# B&R Automation Studio project brdkViLibs
Automation Studio 4.9.4.92 SP; technology packages: mapp 5.20.0, mappView 5.20.0, mappVision 5.20.0

## Configuration ARM

CPU X90CP174.24-00, AutomationRuntime C4.90, Build 6.3.0, Safety 0.0, Vc V4.72.2

CPU X20CP0483, AutomationRuntime C4.90, Build 6.3.0, Safety 0.0, Vc V4.72.2

CPU X20CP0484-1, AutomationRuntime C4.90, Build 6.3.0, Safety 0.0, Vc V4.72.2

### Task classes (Cpu.sw)
```
Cyclic#2 (cycle 20000 us, tolerance 20000 us):
  Demo <- Demo.prg
  Recipe <- Recipe.prg
Binaries: udbdef, mvLoader, TCData, FWRules, TCLang, visionUnit, ashwac, Settings, User, sysconf, viComp, asfw, arconfig, ashwd, iomap, Role, viApp, Config, px, TC, arflatprv, arcoal, arsvcreg, mCoWebSc, Settings_1
Libraries: ViBase, MpRecipe, MpBase, runtime, astime, AsZip, FileIO, AsARCfg, powerlnk, AsEPL, AsIO, sys_lib, standard, MTLinAlg, brdkViMapp, brdkViImg, brdkViGeom, brdkViBase, brdkViVF, brdkViCal, AsTCP, brsystem, AsHttp, AsIecCon, asbrstr, asiodiag, arssl
```

### Task classes (Cpu.sw)
```
Cyclic#1 (cycle 1000 us, tolerance 10000 us):
  Recipe <- Recipe.prg
  Calibratio <- Calibration.prg
Binaries: udbdef, mvLoader, TCData, FWRules, TCLang, ashwac, Settings, User, sysconf, viComp, asfw, arconfig, ashwd, iomap, Role, viApp, Config, px, TC, arflatprv, arcoal, arsvcreg
Libraries: ViBase, MpRecipe, MpBase, runtime, astime, AsZip, FileIO, AsARCfg, powerlnk, AsEPL, AsIO, sys_lib, AsHttp, standard, MTLinAlg, brdkViMapp, brdkViBase, brdkViVF, BRSE_RTK, brdkViCal, brdkViImg, asieccon, brdkViGeom
```

### Task classes (Cpu.sw)
```
Cyclic#1 (cycle 1000 us, tolerance 10000 us):
  Recipe <- Recipe.prg
  Calibratio <- Calibration.prg
Binaries: udbdef, mvLoader, TCData, FWRules, TCLang, ashwac, Settings, User, sysconf, viComp, asfw, arconfig, ashwd, iomap, Role, viApp, Config, px, TC, arflatprv, arcoal, arsvcreg
Libraries: ViBase, MpRecipe, MpBase, brdkViGeom, runtime, astime, AsZip, FileIO, AsARCfg, powerlnk, AsEPL, AsIO, sys_lib, AsHttp, standard, brdkViImg, MTLinAlg, brdkViMapp, AsIODiag, brdkViBase, brdkViVF, BRSE_RTK, brdkViCal, asieccon
```

### Hardware
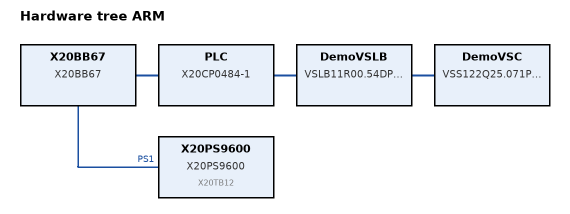
```
DemoVSC : VSS122Q25.071P-000 v1.7.0.606  [PLK1 -> DemoVSLB.PLK2 (NodeNumber=6) [Cable Type=PowerlinkCable, Length=10, Version=1.0.0.3]]
  Supervision = off
  VisionConfig = gBlobCamera
DemoVSLB : VSLB11R00.54DP-000 v1.1.0.323  [PLK1 -> PLC.IF3 (NodeNumber=2) [Cable Type=PowerlinkCable, Length=10, Version=1.0.0.3]; PLK2 -> DemoVSC.PLK1 (NodeNumber=2) [Cable Type=PowerlinkCable, Length=10, Version=1.0.0.3]]
  Supervision = off
  VisionConfig = gBlobCamera
PLC : X20CP0484-1 v1.7.0.0  [SL -> X20BB67.SL1]
  Connector IF2:
    ActivateDevice = 1
    Mode = Manual
    InternetAddress = 192.168.87.210
    SubnetMask = 255.255.255.0
  Connector IF3:
    MtuSize = 1500
    DNAConfiguration = manual
    CycleTime = 1000
    AsyncTimeout = 20
    AsyncSlotsPerCycle = 7
    InternetAddress = 192.168.200.240
    SubnetMask = 255.255.255.0
  ConfigurationID = brdkVision
  UserPartitionSize = 100
  TimerDeviceType = EPLX2X
  TimerDevice = PLC.IF3
  IdleTaskClass = 4
  TaskClassIdleTime = 2000
  Cyclic1Duration = 1000
  Cyclic1Tolerance = 10000
  Cyclic1Stack = 1000000
  Cyclic2Duration = 20000
  Cyclic2Tolerance = 20000
  Cyclic3Duration = 50000
  Cyclic3Tolerance = 50000
  Cyclic4Duration = 100000
  Cyclic4Tolerance = 100000
  Cyclic5Duration = 200000
  Cyclic5Tolerance = 200000
  Cyclic6Duration = 500000
  Cyclic6Tolerance = 500000
  Cyclic7Duration = 1000000
  Cyclic7Tolerance = 1000000
  Cyclic8Duration = 10000
  Cyclic8Tolerance = 30000000
  FileDevice1
  FileDeviceName1 = RECIPE
  FileDevicePath1 = F:\
  FileDevice2
  FileDeviceName2 = SIM
  FileDevicePath2 = C:\simPlc\brdkVision
  FtpUser1
  FtpUsername1 = admin
  FtpUserPassword1 = 4WFXWDK5TMVpfeai37B+7WhwHoefN0SDX+8eS6SXEy0=
  FtpUserSalt1 = PfytuFsU
  FTPAccessRight1 = 0
  FTPdevice1 = ALL
  ActivateOpcUa = 1
  OpcUaInformationModels_PV_Version = 1
X20BB67 : X20BB67 v1.2.0.0
X20PS9600 : X20PS9600 v1.6.0.0  [PS -> X20BB67.PS1; SS1 -> X20TB12.SS]
X20TB12 : X20TB12 v1.0.0.0
```

### Cpu.sw.bak1 - PLC/Cpu.sw.bak1
```
SwConfiguration (CpuAddress=SL1)
  TaskClass Cyclic#1
  TaskClass Cyclic#2:
    Task Demo (Source=Demo.prg, Memory=UserROM, Language=IEC, Debugging=true)
    Task Recipe (Source=Recipe.prg, Memory=UserROM, Language=IEC, Debugging=true)
  TaskClass Cyclic#3
  TaskClass Cyclic#4
  TaskClass Cyclic#5
  TaskClass Cyclic#6
  TaskClass Cyclic#7
  TaskClass Cyclic#8
  Binaries:
    BinaryObject udbdef (Source=, Memory=UserROM, Language=Binary)
    BinaryObject mvLoader (Source=, Memory=UserROM, Language=Binary)
    BinaryObject TCData (Source=, Memory=SystemROM, Language=Binary)
    BinaryObject FWRules (Source=, Memory=UserROM, Language=Binary)
    BinaryObject TCLang (Source=, Memory=UserROM, Language=Binary)
    BinaryObject visionUnit (Source=, Memory=UserROM, Language=Binary)
    BinaryObject arflatprv (Source=, Memory=UserROM, Language=Binary)
    BinaryObject arcoal (Source=, Memory=UserROM, Language=Binary)
    BinaryObject arsvcreg (Source=, Memory=UserROM, Language=Binary)
    BinaryObject mCoWebSc (Source=, Memory=UserROM, Language=Binary)
    BinaryObject ashwac (Source=, Memory=UserROM, Language=Binary)
    BinaryObject Settings (Source=, Memory=UserROM, Language=Binary)
    BinaryObject User (Source=, Memory=UserROM, Language=Binary)
    BinaryObject sysconf (Source=, Memory=SystemROM, Language=Binary)
    BinaryObject viComp (Source=, Memory=UserROM, Language=Binary)
    BinaryObject asfw (Source=, Memory=SystemROM, Language=Binary)
    BinaryObject arconfig (Source=, Memory=SystemROM, Language=Binary)
    BinaryObject ashwd (Source=, Memory=SystemROM, Language=Binary)
    BinaryObject iomap (Source=, Memory=UserROM, Language=Binary)
    BinaryObject Role (Source=, Memory=UserROM, Language=Binary)
    BinaryObject viApp (Source=, Memory=UserROM, Language=Binary)
    BinaryObject Config (Source=, Memory=UserROM, Language=Binary)
    BinaryObject px (Source=, Memory=UserROM, Language=Binary)
    BinaryObject TC (Source=, Memory=UserROM, Language=Binary)
    BinaryObject Settings_1 (Source=, Memory=UserROM, Language=Binary)
  Libraries:
    LibraryObject ViBase (Source=Libraries.ViBase.lby, Memory=UserROM, Language=binary, Debugging=true)
    LibraryObject MpRecipe (Source=Libraries.MpRecipe.lby, Memory=UserROM, Language=Binary, Debugging=true)
    LibraryObject MpBase (Source=Libraries.MpBase.lby, Memory=UserROM, Language=Binary, Debugging=true)
    LibraryObject runtime (Source=Libraries.runtime.lby, Memory=UserROM, Language=binary, Debugging=true)
    LibraryObject astime (Source=Libraries.astime.lby, Memory=UserROM, Language=binary, Debugging=true)
    LibraryObject AsZip (Source=Libraries.AsZip.lby, Memory=UserROM, Language=binary, Debugging=true)
    LibraryObject FileIO (Source=Libraries.FileIO.lby, Memory=UserROM, Language=binary, Debugging=true)
    LibraryObject AsARCfg (Source=Libraries.AsARCfg.lby, Memory=UserROM, Language=binary, Debugging=true)
    LibraryObject powerlnk (Source=Libraries.powerlnk.lby, Memory=UserROM, Language=binary, Debugging=true)
    LibraryObject AsEPL (Source=Libraries.AsEPL.lby, Memory=UserROM, Language=binary, Debugging=true)
    LibraryObject AsIO (Source=Libraries.AsIO.lby, Memory=UserROM, Language=binary, Debugging=true)
    LibraryObject sys_lib (Source=Libraries.sys_lib.lby, Memory=UserROM, Language=binary, Debugging=true)
    LibraryObject standard (Source=Libraries.standard.lby, Memory=UserROM, Language=binary, Debugging=true)
    LibraryObject MTLinAlg (Source=Libraries.MTLinAlg.lby, Memory=UserROM, Language=Binary, Debugging=true)
    LibraryObject brdkViMapp (Source=Libraries.brdkViLibs.brdkViMapp.lby, Memory=UserROM, Language=Binary, Debugging=true)
    LibraryObject brdkViImg (Source=Libraries.brdkViLibs.brdkViImg.lby, Memory=UserROM, Language=Binary, Debugging=true)
    LibraryObject brdkViGeom (Source=Libraries.brdkViLibs.brdkViGeom.lby, Memory=UserROM, Language=Binary, Debugging=true)
    LibraryObject brdkViBase (Source=Libraries.brdkViLibs.brdkViBase.lby, Memory=UserROM, Language=Binary, Debugging=true)
    LibraryObject brdkViVF (Source=Libraries.brdkViLibs.brdkViVF.lby, Memory=UserROM, Language=Binary, Debugging=true)
    LibraryObject brdkViCal (Source=Libraries.brdkViLibs.brdkViCal.lby, Memory=UserROM, Language=Binary, Debugging=true)
    LibraryObject AsTCP (Source=Libraries.AsTCP.lby, Memory=UserROM, Language=binary, Debugging=true)
    LibraryObject brsystem (Source=Libraries.brsystem.lby, Memory=UserROM, Language=binary, Debugging=true)
    LibraryObject AsHttp (Source=Libraries.AsHttp.lby, Memory=UserROM, Language=binary, Debugging=true)
    LibraryObject JSON_WS (Source=Libraries.brdkViLibs.JSON_WS.lby, Memory=UserROM, Language=ANSIC, Debugging=true)
    LibraryObject AsIecCon (Source=Libraries.AsIecCon.lby, Memory=UserROM, Language=binary, Debugging=true)
    LibraryObject arssl (Source=, Memory=UserROM, Language=Binary, Debugging=true)
    LibraryObject asbrstr (Source=, Memory=UserROM, Language=Binary, Debugging=true)
    LibraryObject asiodiag (Source=, Memory=UserROM, Language=Binary, Debugging=true)
```

### IoMap.iom - PLC/IoMap.iom
```iecst
VAR_CONFIG
	::Demo:hw.cam.in.common.moduleOk AT %IX."DemoVSC".ModuleOk;
	::Demo:hw.cam.in.common.serialNumber AT %ID."DemoVSC".SerialNumber;
	::Demo:hw.cam.in.common.moduleId AT %ID."DemoVSC".ModuleID;
	::Demo:hw.cam.in.common.hardwareVariant AT %ID."DemoVSC".HardwareVariant;
	::Demo:hw.cam.in.common.firmwareVersion AT %ID."DemoVSC".FirmwareVersion;
	::Demo:hw.cam.in.status.sensorTemperature AT %IB."DemoVSC".SensorTemperature;
	::Demo:hw.cam.in.status.lightWarningCnt AT %IB."DemoVSC".LightWarningCnt;
	::Demo:hw.cam.in.status.cameraStatus AT %ID."DemoVSC".CameraStatus;
	::Demo:hw.cam.in.status.acceptedAcquisitionCnt AT %IB."DemoVSC".AcceptedAcquisitionCnt;
	::Demo:hw.cam.in.status.completedAcquisitionCnt AT %IB."DemoVSC".CompletedAcquisitionCnt;
	::Demo:hw.cam.in.status.failedAcquisitionCnt AT %IB."DemoVSC".FailedAcquisitionCnt;
	::Demo:hw.cam.in.status.gainLevel AT %IB."DemoVSC".ReadGainLevel;
	::Demo:hw.cam.in.status.focus AT %IW."DemoVSC".ReadFocus;
	::Demo:hw.cam.in.status.exposureTime AT %ID."DemoVSC".ReadExposureTime;
	::Demo:hw.cam.in.status.undervoltageError AT %IX."DemoVSC".UndervoltageError;
	::Demo:hw.cam.in.status.digitalInput AT %IX."DemoVSC".DigitalInput01;
	::Demo:hw.cam.in.status.digitalOutputStatus AT %IX."DemoVSC".DigitalOutputStatus01;
	::Demo:hw.cam.in.status.imageAcquisitionReady AT %IX."DemoVSC".ImageAcquisitionReady;
	::Demo:hw.cam.in.status.imageProcessingActive AT %IX."DemoVSC".ImageProcessingActive;
	::Demo:hw.cam.in.status.cameraProcessingTime AT %IW."DemoVSC".CameraProcessingTime;
	::Demo:hw.cam.in.status.imageProcessingError AT %IW."DemoVSC".ImageProcessingError;
	::Demo:hw.cam.in.status.imageNettime AT %ID."DemoVSC".ImageNettime;
	::Demo:hw.cam.out.par.statusLED AT %QB."DemoVSC".StatusLED;
	::Demo:hw.cam.out.par.gainLevel AT %QB."DemoVSC".GainLevel;
	::Demo:hw.cam.out.par.focus AT %QW."DemoVSC".SetFocus;
	::Demo:hw.cam.out.par.exposureTime AT %QD."DemoVSC".ExposureTime01;
	::Demo:hw.cam.out.par.delayNetTime AT %QD."DemoVSC".DelayNettime01;
	::Demo:hw.cam.out.par.flashColor AT %QB."DemoVSC".FlashColor01;
	::Demo:hw.cam.out.par.flashSegment AT %QB."DemoVSC".FlashSegment01;
	::Demo:hw.cam.out.cmd.digitalOutput AT %QX."DemoVSC".DigitalOutput01;
	::Demo:hw.cam.out.par.IRFilter AT %QX."DemoVSC".IRFilter;
	::Demo:hw.cam.out.par.chromaticLock AT %QX."DemoVSC".ChromaticLock;
	::Demo:hw.cam.out.cmd.searchAcquisitonSettings AT %QX."DemoVSC".SearchAcquisitionSettings;
	::Demo:hw.cam.out.cmd.resetAcquisiton AT %QX."DemoVSC".ResetAcquisition;
	::Demo:hw.cam.out.cmd.imageAcquisition AT %QX."DemoVSC".ImageAcquisition;
	::Demo:hw.blob.out.common.enable AT %QX."DemoVSC".Enable_1;
	::Demo:hw.blob.out.common.numSearchMax AT %QB."DemoVSC".NumSearchMax_1;
	::Demo:hw.blob.out.regionFeatures AT %QX."DemoVSC".RegionFeatures_1;
	::Demo:hw.blob.out.enhancedBlobInformation AT %QX."DemoVSC".EnhancedBlobInformation_1;
	::Demo:hw.blob.out.common.alignment AT %QB."DemoVSC".Alignment_1;
	::Demo:hw.blob.out.common.offsetROI.x AT %QD."DemoVSC".OffsetROIX_1;
	::Demo:hw.blob.out.common.offsetROI.y AT %QD."DemoVSC".OffsetROIY_1;
	::Demo:hw.blob.out.common.offsetROI.orientation AT %QW."DemoVSC".OffsetROIOrientation_1;
	::Demo:hw.blob.out.common.offsetROI.x AT %QD."DemoVSC".OffsetROIRotCenterX_1;
	::Demo:hw.blob.out.common.offsetROI.y AT %QD."DemoVSC".OffsetROIRotCenterY_1;
	::Demo:hw.blob.in.common.numResults AT %IB."DemoVSC".NumResults_1;
	::Demo:hw.blob.in.common.functionProcessingTime AT %IW."DemoVSC".FunctionProcessingTime_1;
	::Demo:hw.blob.in.results[0].modelNumber AT %IB."DemoVSC".ModelNumber_101;
	::Demo:hw.blob.in.results[0].meanGreyValue AT %IB."DemoVSC".MeanGrayValue_101;
	::Demo:hw.blob.in.results[0].clipped AT %IX."DemoVSC".Clipped_101;
	::Demo:hw.blob.in.results[0].area AT %ID."DemoVSC".Area_101;
	::Demo:hw.blob.in.results[0].length AT %ID."DemoVSC".Length_101;
	::Demo:hw.blob.in.results[0].width AT %ID."DemoVSC".Width_101;
	::Demo:hw.blob.in.results[0].xMin AT %ID."DemoVSC".Xmin_101;
	::Demo:hw.blob.in.results[0].xMax AT %ID."DemoVSC".Xmax_101;
	::Demo:hw.blob.in.results[0].yMin AT %ID."DemoVSC".Ymin_101;
	::Demo:hw.blob.in.results[0].yMax AT %ID."DemoVSC".Ymax_101;
	::Demo:hw.blob.in.results[0].circularity AT %IB."DemoVSC".Circularity_101;
	::Demo:hw.blob.in.results[0].rectangularity AT %IB."DemoVSC".Rectangularity_101;
	::Demo:hw.blob.in.results[0].anisometry AT %IW."DemoVSC".Anisometry_101;
	::Demo:hw.blob.in.results[0].innterCirclePositionX AT %ID."DemoVSC".InnerCirclePositionX_101;
	::Demo:hw.blob.in.results[0].innterCirclePositionY AT %ID."DemoVSC".InnerCirclePositionY_101;
	::Demo:hw.blob.in.results[0].innterCircleRadius AT %ID."DemoVSC".InnerCircleRadius_101;
	::Demo:hw.blob.in.results[0].positionX AT %ID."DemoVSC".PositionX_101;
	::Demo:hw.blob.in.results[0].positionY AT %ID."DemoVSC".PositionY_101;
	::Demo:hw.blob.in.results[0].orientation AT %IW."DemoVSC".Orientation_101;
	::Demo:hw.blob.in.results[0].rotCenterX AT %ID."DemoVSC".RotCenterX_101;
	::Demo:hw.blob.in.results[0].rotCenterY AT %ID."DemoVSC".RotCenterY_101;
	::Demo:hw.blob.in.results[1].modelNumber AT %IB."DemoVSC".ModelNumber_102;
	::Demo:hw.blob.in.results[1].meanGreyValue AT %IB."DemoVSC".MeanGrayValue_102;
	::Demo:hw.blob.in.results[1].clipped AT %IX."DemoVSC".Clipped_102;
	::Demo:hw.blob.in.results[1].area AT %ID."DemoVSC".Area_102;
	::Demo:hw.blob.in.results[1].length AT %ID."DemoVSC".Length_102;
	::Demo:hw.blob.in.results[1].width AT %ID."DemoVSC".Width_102;
	::Demo:hw.blob.in.results[1].xMin AT %ID."DemoVSC".Xmin_102;
	::Demo:hw.blob.in.results[1].xMax AT %ID."DemoVSC".Xmax_102;
	::Demo:hw.blob.in.results[1].yMin AT %ID."DemoVSC".Ymin_102;
	::Demo:hw.blob.in.results[1].yMax AT %ID."DemoVSC".Ymax_102;
	::Demo:hw.blob.in.results[1].circularity AT %IB."DemoVSC".Circularity_102;
	::Demo:hw.blob.in.results[1].rectangularity AT %IB."DemoVSC".Rectangularity_102;
	::Demo:hw.blob.in.results[1].anisometry AT %IW."DemoVSC".Anisometry_102;
	::Demo:hw.blob.in.results[1].innterCirclePositionX AT %ID."DemoVSC".InnerCirclePositionX_102;
	::Demo:hw.blob.in.results[1].innterCirclePositionY AT %ID."DemoVSC".InnerCirclePositionY_102;
	::Demo:hw.blob.in.results[1].innterCircleRadius AT %ID."DemoVSC".InnerCircleRadius_102;
	::Demo:hw.blob.in.results[1].positionX AT %ID."DemoVSC".PositionX_102;
	::Demo:hw.blob.in.results[1].positionY AT %ID."DemoVSC".PositionY_102;
	::Demo:hw.blob.in.results[1].orientation AT %IW."DemoVSC".Orientation_102;
	::Demo:hw.blob.in.results[1].rotCenterX AT %ID."DemoVSC".RotCenterX_102;
	::Demo:hw.blob.in.results[1].rotCenterY AT %ID."DemoVSC".RotCenterY_102;
	::Demo:hw.blob.in.results[2].modelNumber AT %IB."DemoVSC".ModelNumber_103;
	::Demo:hw.blob.in.results[2].meanGreyValue AT %IB."DemoVSC".MeanGrayValue_103;
	::Demo:hw.blob.in.results[2].clipped AT %IX."DemoVSC".Clipped_103;
	::Demo:hw.blob.in.results[2].area AT %ID."DemoVSC".Area_103;
	::Demo:hw.blob.in.results[2].length AT %ID."DemoVSC".Length_103;
	::Demo:hw.blob.in.results[2].width AT %ID."DemoVSC".Width_103;
	::Demo:hw.blob.in.results[2].xMin AT %ID."DemoVSC".Xmin_103;
	::Demo:hw.blob.in.results[2].xMax AT %ID."DemoVSC".Xmax_103;
	::Demo:hw.blob.in.results[2].yMin AT %ID."DemoVSC".Ymin_103;
	::Demo:hw.blob.in.results[2].yMax AT %ID."DemoVSC".Ymax_103;
	::Demo:hw.blob.in.results[2].circularity AT %IB."DemoVSC".Circularity_103;
	::Demo:hw.blob.in.results[2].rectangularity AT %IB."DemoVSC".Rectangularity_103;
	::Demo:hw.blob.in.results[2].anisometry AT %IW."DemoVSC".Anisometry_103;
	::Demo:hw.blob.in.results[2].innterCirclePositionX AT %ID."DemoVSC".InnerCirclePositionX_103;
	::Demo:hw.blob.in.results[2].innterCirclePositionY AT %ID."DemoVSC".InnerCirclePositionY_103;
	::Demo:hw.blob.in.results[2].innterCircleRadius AT %ID."DemoVSC".InnerCircleRadius_103;
	::Demo:hw.blob.in.results[2].positionX AT %ID."DemoVSC".PositionX_103;
	::Demo:hw.blob.in.results[2].positionY AT %ID."DemoVSC".PositionY_103;
	::Demo:hw.blob.in.results[2].orientation AT %IW."DemoVSC".Orientation_103;
	::Demo:hw.blob.in.results[2].rotCenterX AT %ID."DemoVSC".RotCenterX_103;
	::Demo:hw.blob.in.results[2].rotCenterY AT %ID."DemoVSC".RotCenterY_103;
	::Demo:hw.blob.in.results[3].modelNumber AT %IB."DemoVSC".ModelNumber_104;
	::Demo:hw.blob.in.results[3].meanGreyValue AT %IB."DemoVSC".MeanGrayValue_104;
	::Demo:hw.blob.in.results[3].clipped AT %IX."DemoVSC".Clipped_104;
	::Demo:hw.blob.in.results[3].area AT %ID."DemoVSC".Area_104;
	::Demo:hw.blob.in.results[3].length AT %ID."DemoVSC".Length_104;
	::Demo:hw.blob.in.results[3].width AT %ID."DemoVSC".Width_104;
	::Demo:hw.blob.in.results[3].xMin AT %ID."DemoVSC".Xmin_104;
	::Demo:hw.blob.in.results[3].xMax AT %ID."DemoVSC".Xmax_104;
	::Demo:hw.blob.in.results[3].yMin AT %ID."DemoVSC".Ymin_104;
	::Demo:hw.blob.in.results[3].yMax AT %ID."DemoVSC".Ymax_104;
	::Demo:hw.blob.in.results[3].circularity AT %IB."DemoVSC".Circularity_104;
	::Demo:hw.blob.in.results[3].rectangularity AT %IB."DemoVSC".Rectangularity_104;
	::Demo:hw.blob.in.results[3].anisometry AT %IW."DemoVSC".Anisometry_104;
	::Demo:hw.blob.in.results[3].innterCirclePositionX AT %ID."DemoVSC".InnerCirclePositionX_104;
	::Demo:hw.blob.in.results[3].innterCirclePositionY AT %ID."DemoVSC".InnerCirclePositionY_104;
	::Demo:hw.blob.in.results[3].innterCircleRadius AT %ID."DemoVSC".InnerCircleRadius_104;
	::Demo:hw.blob.in.results[3].positionX AT %ID."DemoVSC".PositionX_104;
	::Demo:hw.blob.in.results[3].positionY AT %ID."DemoVSC".PositionY_104;
	::Demo:hw.blob.in.results[3].orientation AT %IW."DemoVSC".Orientation_104;
	::Demo:hw.blob.in.results[3].rotCenterX AT %ID."DemoVSC".RotCenterX_104;
	::Demo:hw.blob.in.results[3].rotCenterY AT %ID."DemoVSC".RotCenterY_104;
	::Demo:hw.io.input.nettime AT %ID."PLC".IF3.NettimeSoC;
	::Demo:hw.backLight[0].in.common.moduleOk AT %IX."DemoVSLB".ModuleOk;
	::Demo:hw.backLight[0].in.common.serialNumber AT %ID."DemoVSLB".SerialNumber;
	::Demo:hw.backLight[0].in.common.moduleId AT %ID."DemoVSLB".ModuleID;
	::Demo:hw.backLight[0].in.common.hardwareVariant AT %ID."DemoVSLB".HardwareVariant;
	::Demo:hw.backLight[0].in.common.firmwareVersion AT %ID."DemoVSLB".FirmwareVersion;
	::Demo:hw.backLight[0].in.status.ready AT %IX."DemoVSLB".Ready;
	::Demo:hw.backLight[0].in.status.status AT %ID."DemoVSLB".Status;
	::Demo:hw.backLight[0].in.status.acceptedFlashCnt AT %IB."DemoVSLB".AcceptedFlashCnt;
	::Demo:hw.backLight[0].in.status.completedFlashCnt AT %IB."DemoVSLB".CompletedFlashCnt;
	::Demo:hw.backLight[0].in.status.failedFlashCnt AT %IB."DemoVSLB".FailedFlashCnt;
	::Demo:hw.backLight[0].in.status.LightWarningCnt AT %IB."DemoVSLB".LightWarningCnt;
	::Demo:hw.backLight[0].in.status.sensorTemperatureControllerBoard AT %IB."DemoVSLB".SensorTemperature;
	::Demo:hw.backLight[0].out.cmd.flashTrigger AT %QX."DemoVSLB".FlashTrigger;
	::Demo:hw.backLight[0].out.cmd.resetFlashTrigger AT %QX."DemoVSLB".ResetFlashTrigger;
	::Demo:hw.backLight[0].out.par.nettime AT %QD."DemoVSLB".Nettime01;
	::Demo:hw.backLight[0].out.par.exposureTime AT %QD."DemoVSLB".ExposureTime01;
	::Demo:hw.backLight[0].out.par.flashColor AT %QB."DemoVSLB".FlashColor01;
END_VAR
```

### Config.mprecipecsv - PLC/mappServices/Config.mprecipecsv
```
Element gRecipeCsv (Type=mprecipecsv)
```

### IoMap.iom - X20CP0483/IoMap.iom
```iecst
VAR_CONFIG
	::Calibratio:hw.out.focus AT %QW."VSC122R14.033P-000".SetFocus;
	::Calibratio:hw.out.expTime AT %QD."VSC122R14.033P-000".ExposureTime01;
	::Calibratio:hw.out.delayNettime AT %QD."VSC122R14.033P-000".DelayNettime01;
	::Calibratio:hw.out.ledColor AT %QB."VSC122R14.033P-000".FlashColor01;
	::Calibratio:hw.out.ledSegment AT %QB."VSC122R14.033P-000".FlashSegment01;
	::Calibratio:hw.in.ready AT %IX."VSC122R14.033P-000".ImageAcquisitionReady;
	::Calibratio:hw.out.trigger AT %QX."VSC122R14.033P-000".ImageAcquisition;
	::Calibratio:hw.out.irFilter AT %QX."VSC122R14.033P-000".IRFilter;
	::Calibratio:hw.out.enable AT %QX."VSC122R14.033P-000".VF1Enable;
	::Calibratio:hw.out.numMax AT %QB."VSC122R14.033P-000".VF1NumSearchMax;
	::Calibratio:hw.in.imgTime AT %ID."VSC122R14.033P-000".ImageNettime;
	::Calibratio:hw.in.va.numRes AT %IB."VSC122R14.033P-000".NumResults;
	::Calibratio:hw.in.va.res[0].posX AT %ID."VSC122R14.033P-000".PositionX01;
	::Calibratio:hw.in.va.res[1].posX AT %ID."VSC122R14.033P-000".PositionX02;
	::Calibratio:hw.in.va.res[2].posX AT %ID."VSC122R14.033P-000".PositionX03;
	::Calibratio:hw.in.va.res[3].posX AT %ID."VSC122R14.033P-000".PositionX04;
	::Calibratio:hw.in.va.res[0].posY AT %ID."VSC122R14.033P-000".PositionY01;
	::Calibratio:hw.in.va.res[1].posY AT %ID."VSC122R14.033P-000".PositionY02;
	::Calibratio:hw.in.va.res[2].posY AT %ID."VSC122R14.033P-000".PositionY03;
	::Calibratio:hw.in.va.res[3].posY AT %ID."VSC122R14.033P-000".PositionY04;
	::Calibratio:hw.out.delayNettime AT %QD."VSLB11Q00.54DP-000".Nettime01;
	::Calibratio:hw.out.expTime AT %QD."VSLB11Q00.54DP-000".ExposureTime01;
	::Calibratio:hw.out.ledColor AT %QB."VSLB11Q00.54DP-000".FlashColor01;
	::Calibratio:hw.out.trigger AT %QX."VSLB11Q00.54DP-000".FlashTrigger;
	::Calibratio:hw.out.useRegionFeat AT %QX."VSC122R14.033P-000".VF1RegionFeatures;
	::Calibratio:hw.in.nettime AT %ID."X20CP0483".IF3.NettimeSoC;
END_VAR
```

### IoMap.iom - X20CP0484_1/IoMap.iom
```iecst
VAR_CONFIG
	::Calibratio:hw.io.input.nettime AT %ID."X20CP0484_1".IF3.NettimeSoC;
END_VAR
```

### Settings.vicfg - X20CP0484_1/mappVision/Settings.vicfg
```
Element VisionSettings (Type=vicfg)
  ActivateVisualization = TRUE
  FileDeviceName
  Permissions:
    WriteAccessRole = Everyone
```

### viComp.visioncomponent - X20CP0484_1/mappVision/viComp.visioncomponent
```
Element gBlobCamera (Type=visioncomponent)
  VisionApplicationReference = BLOBCam
```

## Configuration Intel

CPU X20CP1586, AutomationRuntime C4.90, Build 6.3.0, Safety 0.0, Vc 

CPU X20CP1586, AutomationRuntime C4.90, Build 6.3.0, Safety 0.0, Vc 

### Task classes (Cpu.sw)
```
Cyclic#1 (cycle 2000 us):
  Recipe <- Recipe.prg
  Demo <- Demo.prg
Binaries: udbdef, mvLoader, TCData, FWRules, TCLang, arflatprv, arcoal, arsvcreg, visionUnit, ashwac, Settings, User, sysconf, viComp, asfw, arconfig, ashwd, iomap, Role, viApp, Config
Libraries: ViBase, MpRecipe, MpBase, MTLinAlg, runtime, astime, AsZip, FileIO, AsARCfg, powerlnk, AsEPL, AsIO, sys_lib, standard, brdkViBase, brdkViMapp, brdkViVF, brdkViCal, AsIODiag, arssl, asieccon
```

### Task classes (Cpu.sw)
```
Cyclic#1 (cycle 2000 us):
  Recipe <- Recipe.prg
  Calibratio <- Calibration.prg
Binaries: udbdef, mvLoader, TCData, FWRules, TCLang, ashwac, Settings, User, sysconf, viComp, asfw, arconfig, ashwd, iomap, Role, viApp, Config, arflatprv, arcoal, arsvcreg
Libraries: ViBase, MpRecipe, MpBase, MTLinAlg, runtime, astime, AsZip, FileIO, AsARCfg, powerlnk, AsEPL, AsIO, sys_lib, AsHttp, standard, arssl, brdkViBase, brdkViGeom, brdkViImg, brdkViMapp, brdkViVF, BRSE_RTK, brdkViCal
```

### Hardware
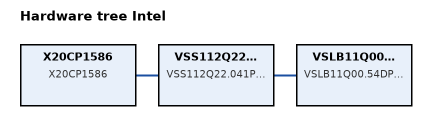
```
VSLB11Q00.54DP-000 : VSLB11Q00.54DP-000 v1.1.0.323  [PLK1 -> VSS112Q22.041P-000.PLK2 (NodeNumber=2) [Cable Type=PowerlinkCable, Length=10, Version=1.0.0.3]]
  VisionConfig = gBlobCamera
VSS112Q22.041P-000 : VSS112Q22.041P-000 v1.5.0.489  [PLK1 -> X20CP1586.IF3 (NodeNumber=1) [Cable Type=PowerlinkCable, Length=10, Version=1.0.0.3]; PLK2 -> VSLB11Q00.54DP-000.PLK1 (NodeNumber=1) [Cable Type=PowerlinkCable, Length=10, Version=1.0.0.3]]
  Supervision = off
  VisionConfig = gBlobCamera
X20CP1586 : X20CP1586 v1.8.1.0
  Connector IF2:
    ActivateDevice = 1
    Mode = Manual
    InternetAddress = 192.168.87.212
    SubnetMask = 255.255.255.0
  Connector IF3:
    MtuSize = 1500
    CycleTime = 400
    InternetAddress = 192.168.200.240
    SubnetMask = 255.255.255.0
  ConfigurationID = BilwincoHMI
  UserPartitionSize = 50
  ApplicationStorageType = NORMAL
  Cyclic1Duration = 2000
  FileDevice1
  FileDeviceName1 = RECIPE
  FileDevicePath1 = D:\
  FtpUser1
  FtpUsername1 = admin
  FtpUserPassword1 = +uX37b/Iy9gDw18lRrZX7EcbwYFwQWpAJkuUgOjAEQo=  // admin
  FtpUserSalt1 = ij+K1uf1
  FTPAccessRight1 = 0
  FTPdevice1 = ALL
  ActivateOpcUa = 1
  OpcUaInformationModels_PV_Version = 1
```

### IoMap.iom - PLC/IoMap.iom
```iecst
VAR_CONFIG
	::Demo:hw.io.input.nettime AT %ID."X20CP1586".IF3.NettimeSoC;
END_VAR
```

- Safety project (password-protected, skipped)

### IoMap.iom - X20CP1586/IoMap.iom
```iecst
VAR_CONFIG
	::Calibratio:hw.out.focus AT %QW."VSS112Q22.041P-000".SetFocus;
	::Calibratio:hw.out.expTime AT %QD."VSS112Q22.041P-000".ExposureTime01;
	::Calibratio:hw.out.delayNettime AT %QD."VSS112Q22.041P-000".DelayNettime01;
	::Calibratio:hw.out.ledColor AT %QB."VSS112Q22.041P-000".FlashColor01;
	::Calibratio:hw.out.ledSegment AT %QB."VSS112Q22.041P-000".FlashSegment01;
	::Calibratio:hw.in.ready AT %IX."VSS112Q22.041P-000".ImageAcquisitionReady;
	::Calibratio:hw.out.trigger AT %QX."VSS112Q22.041P-000".ImageAcquisition;
	::Calibratio:hw.out.irFilter AT %QX."VSS112Q22.041P-000".IRFilter;
	::Calibratio:hw.out.enable AT %QX."VSS112Q22.041P-000".VF1Enable;
	::Calibratio:hw.out.numMax AT %QB."VSS112Q22.041P-000".VF1NumSearchMax;
	::Calibratio:hw.in.imgTime AT %ID."VSS112Q22.041P-000".ImageNettime;
	::Calibratio:hw.in.va.numRes AT %IB."VSS112Q22.041P-000".NumResults;
	::Calibratio:hw.in.va.res[0].posX AT %ID."VSS112Q22.041P-000".PositionX01;
	::Calibratio:hw.in.va.res[1].posX AT %ID."VSS112Q22.041P-000".PositionX02;
	::Calibratio:hw.in.va.res[2].posX AT %ID."VSS112Q22.041P-000".PositionX03;
	::Calibratio:hw.in.va.res[3].posX AT %ID."VSS112Q22.041P-000".PositionX04;
	::Calibratio:hw.in.va.res[0].posY AT %ID."VSS112Q22.041P-000".PositionY01;
	::Calibratio:hw.in.va.res[1].posY AT %ID."VSS112Q22.041P-000".PositionY02;
	::Calibratio:hw.in.va.res[2].posY AT %ID."VSS112Q22.041P-000".PositionY03;
	::Calibratio:hw.in.va.res[3].posY AT %ID."VSS112Q22.041P-000".PositionY04;
	::Calibratio:hw.out.delayNettime AT %QD."VSLB11Q00.54DP-000".Nettime01;
	::Calibratio:hw.out.expTime AT %QD."VSLB11Q00.54DP-000".ExposureTime01;
	::Calibratio:hw.out.ledColor AT %QB."VSLB11Q00.54DP-000".FlashColor01;
	::Calibratio:hw.out.trigger AT %QX."VSLB11Q00.54DP-000".FlashTrigger;
	::Calibratio:hw.in.nettime AT %ID."X20CP1586".IF3.NettimeSoC;
	::Calibratio:hw.out.useRegionFeat AT %QX."VSS112Q22.041P-000".VF1RegionFeatures;
END_VAR
```

## Logical view

Binary libraries used (declarations not repeated): operator, runtime, astime, AsIecCon, AsZip, FileIO, AsARCfg, powerlnk, AsEPL, AsIO, sys_lib, AsHttp, standard, AsBrStr, AsMem, brdkViMapp 1.00.0, brdkViBase 1.00.0, brdkViGeom 1.00.0, brdkViImg 1.00.0, brdkViVF 1.00.0, BRSE_RTK 1.04.0, MTLinAlg 5.17.0, brdkViCal 1.00.0, ViBase 5.16.1, MpRecipe 5.20.0, MpBase 5.20.0, brdkViGeom 1.00.1, brdkViImg 5.20.0, brdkViVF, brdkViBase 1.00.0, brdkViMapp, brdkViCal, brdkViMapp 1.01.0, brdkViBase, brdkViVF, brdkViCal, brdkViImg 5.20.1, brdkViGeom

### Global.typ - Global data types
```iecst
TYPE
	gVisionCtrl_type : STRUCT
		Cmd : gVisionCtrlPar_type;
		Parameters : gVisionCtrlPar_type;
		Status : gVisionCtrlStatus_type;
	END_STRUCT;
	gVisionCtrlCmd_type : STRUCT
		ImageAcquisition : BOOL;
		ImageProcessingActive : BOOL;
		SearchAcquisitionSettings : BOOL;
		Enable : BOOL;
	END_STRUCT;
	gVisionCtrlPar_type : STRUCT
		FlashColor : USINT;
		FlashSegment : USINT;
		SetFocus : UINT;
		ExposureTime : UDINT;
		NumSearchMax : USINT;
		Nettime : DINT;
		DelayNettime : DINT;
	END_STRUCT;
	gVisionCtrlStatus_type : STRUCT
		Status : USINT;
		CameraStatus : UDINT;
	END_STRUCT;
END_TYPE
```

### Package Logical/Libraries - Global libraries

### Global.var - Global variables
```iecst
VAR
	gVisionCtrl : gVisionCtrl_type;
END_VAR

VAR CONSTANT

END_VAR
```

- Visualisation Logical/mappView (not shown)

- brdkByReference.py (not shown)

### Program Logical/Recipe (IEC)

#### Types.typ
```iecst
TYPE
	recipe_typ : 	STRUCT
		VF : brdkViMapp_VF_typ;
	END_STRUCT;
END_TYPE
```

#### Variables.var
```iecst
VAR
	save : BOOL;
	load : BOOL;
	recipe : recipe_typ;
	mpRecipe : MpRecipeCsv;
	error : STRING[200];
	mpRecipeUIStruct : MpRecipeUIConnectType;
	mpRecipeUI : MpRecipeUI;
	viBaseLoadVa : ViBaseLoadApplication;
	mpRecipeRegPar : MpRecipeRegParSync;
	oldLoadedRecipe : STRING[255];
	viLoadVA : USINT;
END_VAR
```

#### Main.st
```iecst
PROGRAM _INIT
	(* Insert code here *)
	mpRecipe.Enable := TRUE;
	mpRecipe.DeviceName := ADR('RECIPE');
	mpRecipe.FileName := ADR('reicpe.csv');
	mpRecipe.MpLink := ADR(gRecipeCsv);
	mpRecipe();

	mpRecipeUI.Enable := TRUE;
	mpRecipeUI.MpLink := ADR(gRecipeCsv);
	mpRecipeUI.UIConnect := ADR(mpRecipeUIStruct);
	mpRecipeUI();

	mpRecipeRegPar.Enable := TRUE;
	mpRecipeRegPar.MpLink := ADR(gRecipeCsv);
	mpRecipeRegPar.PVName := ADR('::Recipe:recipe');
	mpRecipeRegPar();

END_PROGRAM

PROGRAM _CYCLIC
	(* Insert code here *)

	// Perhaps not the best way to detect if a new recipe is loaded but it works as long as its not the same recipe :)
	mpRecipe.UpdateNotification := mpRecipe.Info.LastLoadedRecipe <> oldLoadedRecipe;
	oldLoadedRecipe := mpRecipe.Info.LastLoadedRecipe;

	// wait for Mapp Recipe save notification
	IF mpRecipeRegPar.SaveNotification THEN
		// Get VF information from AR config system
		brdkViMapp_getVfDataSet('BLOBCam',1,ADR(recipe.VF.params),ADR(recipe.VF.ROI),ADR(recipe.VF.widgetModels),SIZEOF(recipe.VF.ROI),ADR(error));
		// Allow MpRecipe to save recipe to file
		mpRecipeRegPar.ConfirmSave := TRUE;
	END_IF

	// wait for Mapp Recipe update notification
	IF mpRecipeRegPar.UpdateNotification THEN
		// Set VF info into AR config system
		brdkViMapp_setVfDataSet('BLOBCam',1,ADR(recipe.VF.params),ADR(recipe.VF.ROI),ADR(recipe.VF.widgetModels),ADR(error));
		//Trigger a Load of the VA from AS config system down to the camera
		viBaseLoadVa.Execute := TRUE;
		viBaseLoadVa.MpLink := ADR(gBlobCamera);
		viBaseLoadVa.Name := ADR('BLOBCam');
	END_IF

	// Check if load of VA to camera is done
	IF viBaseLoadVa.Done OR viBaseLoadVa.Error THEN
		viBaseLoadVa.Execute := FALSE;
	END_IF

	// FB calls
	mpRecipe();
	mpRecipeUI();
	mpRecipeRegPar();
	viBaseLoadVa();
END_PROGRAM

PROGRAM _EXIT
	(* Insert code here *)
	mpRecipe(Enable := FALSE);
	mpRecipeUI(Enable := FALSE);
	mpRecipeRegPar(Enable := FALSE);

END_PROGRAM
```

### Program Logical/Calibration (IEC)

#### Main.st - Init, cyclic, exit code
```iecst
PROGRAM _INIT
	(* Insert code here *)
	hmi.in.par.expTime := 700;
	hmi.in.par.focus := 411;
	hmi.in.par.LED := 1;

	this.mappView.enable 		:= TRUE;
	this.mappView.cameraIp 		:= '192.168.200.1';
	this.mappView.getImageArray := FALSE;
	this.mappView.timeout 		:= 3000;

	this.mpRecipeRegPar.MpLink := ADR(gRecipeCsv);
	this.mpRecipeRegPar.PVName := ADR('::Calibratio:hmi.in.par');

END_PROGRAM

PROGRAM _CYCLIC
	(* Insert code here *)

	// trigger image
	hw.out.ledColor 	:= hmi.in.par.LED;
	hw.out.ledSegment 	:= hmi.in.par.LEDsegment;
	hw.out.expTime 		:= hmi.in.par.expTime;
	hw.out.focus 		:= hmi.in.par.focus;
	hw.out.irFilter 	:= hw.out.ledColor = 100;

	CASE state OF
		0:
			IF NOT hw.out.trigger  AND hw.in.ready THEN
				IF hmi.in.cmd.calibrate THEN
					// for calibration we only look for 4 round Blobs
					hw.out.numMax := 4;
					hw.out.enable := TRUE;
					hw.out.useRegionFeat := TRUE;

					state := 10;
				ELSIF hmi.in.cmd.trigger THEN
					hw.out.enable := FALSE;
					hw.out.useRegionFeat := FALSE;
					state := 10;
				END_IF
			END_IF

		10:
			// trigger image with nettime
			hw.out.trigger := TRUE;
			hw.out.delayNettime := hw.in.nettime+ 20000;
			this.timeoutTrigger.PT := T#2000ms;
			this.timeoutTrigger.IN := TRUE;

			state := 20;

		20:
			// check if a new image is done
			IF hw.in.imgTime <> this.oldTime THEN
				this.oldTime := hw.in.imgTime;
				this.mappView.updateImage := TRUE;

				// check if its a calibration or its a pick result image
				IF hmi.in.cmd.calibrate THEN
					IF hw.in.va.numRes = 4  THEN
						this.calcCalibrate := TRUE;
					END_IF
				ELSE
					this.getPicks := TRUE;
				END_IF

				hmi.in.cmd.trigger := hmi.in.cmd.calibrate := FALSE;
				hw.out.trigger := FALSE;

				state := 0;
			ELSIF this.timeoutTrigger.Q THEN
				state := 0;
				this.timeoutTrigger.IN := hw.out.trigger := FALSE;
				hmi.in.cmd.trigger := hmi.in.cmd.calibrate := FALSE;
				hw.out.trigger := FALSE;
			END_IF

	END_CASE
	this.timeoutTrigger();

	// Process the picks
	IF this.getPicks THEN
		this.getPicks := FALSE;

		// reset current results
		brsmemset(ADR(this.matchRes),0,SIZEOF(this.matchRes));
		hmi.out.overlay := '';

		// Process each result from the VF
		FOR i:= 0 TO hw.in.VA_match.numRes BY 1 DO

			// convert to decimal numbers (and offset andge)
			this.matchRes[i].imgPos.x := DINT_TO_REAL(hw.in.VA_match.res[i].posX) / 100.0;
			this.matchRes[i].imgPos.y := DINT_TO_REAL(hw.in.VA_match.res[i].posX) / 100.0;
			this.matchRes[i].angle := DINT_TO_REAL(hw.in.VA_match.res[i].angle) / 100.0 + hmi.in.par.offset.z;

			// find rotation point (will be used to add offset to x and y axis relative to object orientation)
			this.rotPoint.x := COS(this.matchRes[i].angle*0.0174532925199444);
			this.rotPoint.y := SIN(this.matchRes[i].angle*-0.0174532925199444);
			// add offset (x,y) to object poisition relative to object orientation
			this.matchRes[i].imgPos.x := this.matchRes[i].imgPos.x  + this.rotPoint.x*hmi.in.par.offset.x + this.rotPoint.y*hmi.in.par.offset.y;
			this.matchRes[i].imgPos.y := this.matchRes[i].imgPos.y  + this.rotPoint.y*hmi.in.par.offset.x - this.rotPoint.x*hmi.in.par.offset.y;

			// Get 3d position
			brdkViCal_2dTo3d(this.matchRes[i].imgPos,this.invP,this.matchRes[i].pickPos); // Project px to mm
			this.matchRes[i].pickPos.z := LREAL_TO_REAL(brdkViCal_2dto3dOrientation(this.matchRes[i].angle,this.invP,this.imgCenter.x,this.imgCenter.y));

			// offset shape point to result location
			IF this.shapesPx.clearenceEnd.numPoints > 0 THEN
				FOR j:=0 TO this.shapesPx.clearenceEnd.numPoints - 1 BY 1 DO
					brdkViGeom_offsetVector(-this.matchRes[i].angle, this.matchRes[i].imgPos,this.matchRes[i].shapePoints.clearenceEnd[j]);
				END_FOR
				brdkViGeom_drawSvgPoly(this.matchRes[i].shapePoints.clearenceEnd[0],this.shapesPx.clearenceEnd.numPoints, ADR(hmi.out.overlay),ADR('style="fill:yellow;stroke:yellow;stroke-width:5;fill-opacity:0.3;stroke-opacity:1"'));
			END_IF

			IF this.shapesPx.clearenceStart.numPoints > 0 THEN
				FOR j:=0 TO this.shapesPx.clearenceStart.numPoints - 1 BY 1 DO
					brdkViGeom_offsetVector(-this.matchRes[i].angle, this.matchRes[i].imgPos,this.matchRes[i].shapePoints.clearenceStart[j]);
				END_FOR
				brdkViGeom_drawSvgPoly(this.matchRes[i].shapePoints.clearenceStart[0],this.shapesPx.clearenceStart.numPoints, ADR(hmi.out.overlay),ADR('style="fill:yellow;stroke:yellow;stroke-width:5;fill-opacity:0.3;stroke-opacity:1"'));
			END_IF

			IF this.shapesPx.reference.numPoints > 0 THEN
				FOR j:=0 TO this.shapesPx.reference.numPoints - 1 BY 1 DO
					brdkViGeom_offsetVector(-this.matchRes[i].angle, this.matchRes[i].imgPos,this.matchRes[i].shapePoints.reference[j]);
				END_FOR
				brdkViGeom_drawSvgPoly(this.matchRes[i].shapePoints.reference[0],this.shapesPx.reference.numPoints, ADR(hmi.out.overlay),ADR('style="fill:green;stroke:green;stroke-width:5;fill-opacity:0.3;stroke-opacity:1"'));
			END_IF

		END_FOR

	END_IF

	(*
	Calibation Plate

	|-------------------|
	|					| 37,5
	|	O			O	|
	|					| 			 150mm
	|					| 75mm
	|					|
	|	O		 	O	|
	| 					| 37,5mm
	--------------------|
	37,5     75mm    37,5
	_____________________
			150 mm

	Placement of real coordinate systems compared to image and calibration plate holes

	0,0         imgWidth,0
	   /|\ Y
	O	|	O
		|
	----------> X
		|
	O	|	O
		|
	0,imgHeiht	imgWidht,imgHeight
	*)

	// check that we only have 4 results
	IF this.calcCalibrate THEN
		this.calcCalibrate := FALSE;
		// Transfer VA results to 2 image points
		FOR i:=0 TO 3 BY 1 DO
			this.imgPos[i].x := DINT_TO_LREAL(hw.in.va.res[i].posX) /100.0; // px
			this.imgPos[i].y := DINT_TO_LREAL(hw.in.va.res[i].posY) /100.0; // px

			IF this.imgPos[i].x > this.imgWidth/2 THEN
				this.realPos[i].x := 37.5; //mm
			ELSE
				this.realPos[i].x := -37.5; // mm

			END_IF

			IF this.imgPos[i].y > this.imgHeight/2 THEN
				this.realPos[i].y := -37.5; // mm

			ELSE
				this.realPos[i].y := 37.5; //mm
			END_IF

		END_FOR

		brdkViCal_Calibration(this.realPos[0],this.imgPos[0],4,hmi.in.par.P);

		hmi.out.overlay := '';
		brdkViGeom_drawCalibration(hmi.in.par.P,75,this.realPos[0],4,ADR(hmi.out.overlay),ADR('style="fill:blue;stroke:blue;stroke-width:5;fill-opacity:0.3;stroke-opacity:1"'),ADR('style="fill:red;stroke:red;stroke-width:5;fill-opacity:1;stroke-opacity:1"'));

	END_IF

	// Handle image click event
	IF hmi.in.cmd.click THEN
		hmi.in.cmd.click := FALSE;

		this.tmp2D.x := hmi.in.cmd.x;
		this.tmp2D.y := hmi.in.cmd.y;

		// get invers projection matix (only need to be done one time as the projection matrix only changes if a new calibration is done
		brdkViCal_InvP(hmi.in.par.P,this.invP);

		// from image to real coordinates
		brdkViCal_2dTo3d(this.tmp2D,this.invP,hmi.out.realPos);
	END_IF

	this.mappView.imageFormat 	:= hmi.in.par.imgFormat;
	this.mappView.jpegQuality 	:= hmi.in.par.imgQuality;
	this.mappView.pSvgImage 	:= ADR(hmi.out.svg);
	this.mappView.pImageArray 	:= ADR(this.imgArr);
	this.mappView();

	// recipe
	this.mpRecipeRegPar.ConfirmSave := this.mpRecipeRegPar.SaveNotification;
	this.mpRecipeRegPar(Enable := TRUE);

END_PROGRAM

PROGRAM _EXIT
	(* Insert code here *)
	this.mappView(enable := FALSE);
	this.mpRecipeRegPar(Enable := FALSE);
END_PROGRAM
```

#### Types.typ - Local data types
```iecst
TYPE
	match_res_typ : 	STRUCT
		score : USINT;
		angle : INT;
		posY : DINT;
		posX : DINT;
	END_STRUCT;
	blob_res_typ : 	STRUCT
		width : UDINT;
		maxX : DINT;
		minX : DINT;
		length : UDINT;
		posY : DINT;
		posX : DINT;
	END_STRUCT;
	cam_in_match_typ : 	STRUCT
		numRes : USINT;
		res : ARRAY[0..19]OF match_res_typ;
	END_STRUCT;
	cam_in_typ : 	STRUCT
		imgTime : DINT;
		ready : BOOL;
		va : va_res_typ;
		nettime : DINT;
		VA_match : cam_in_match_typ;
	END_STRUCT;
	cam_out_match_typ : 	STRUCT
		maxNum : USINT;
		enable : BOOL;
		timeout : UINT;
		maxOverlap : USINT;
		minScore : USINT;
	END_STRUCT;
	cam_out_typ : 	STRUCT
		expTime : UDINT := 400;
		ledSegment : USINT := 15;
		ledColor : USINT := 100;
		focus : UINT := 150;
		enable : BOOL := TRUE;
		enableEnhanced : BOOL := TRUE;
		numMax : USINT := 4;
		trigger : BOOL;
		irFilter : BOOL;
		delayNettime : DINT;
		useRegionFeat : BOOL;
		VA_match : cam_out_match_typ;
	END_STRUCT;
	cam_typ : 	STRUCT
		out : cam_out_typ;
		in : cam_in_typ;
	END_STRUCT;
	hmi_in_cmd_typ : 	STRUCT
		trigger : BOOL;
		calibrate : BOOL;
		elemId : STRING[80];
		y : REAL;
		x : REAL;
		click : BOOL;
	END_STRUCT;
	hmi_in_typ : 	STRUCT
		cmd : hmi_in_cmd_typ;
		par : recipe_typ;
	END_STRUCT;
	hmi_out_typ : 	STRUCT
		overlay : STRING[20000];
		svg : STRING[6000000];
		realPos : brdkViBase_3d_typ;
	END_STRUCT;
	hmi_typ : 	STRUCT
		in : hmi_in_typ;
		out : hmi_out_typ;
	END_STRUCT;
	hw_typ : 	STRUCT
	END_STRUCT;
	local_typ : 	STRUCT
		realPos : ARRAY[0..3]OF brdkViBase_3d_typ;
		imgPos : ARRAY[0..3]OF brdkViBase_2d_typ;
		invP : ARRAY[0..2,0..2]OF LREAL;
		imgCenter : brdkViBase_2d_typ;
		tmp2D1 : brdkViBase_2d_typ;
		tmp2D : brdkViBase_2d_typ;
		tmp3D : brdkViBase_3d_typ;
		tmpLREAL : LREAL;
		imgHeight : LREAL := 1024;
		imgWidth : LREAL := 1250;
		calcCalibrate : BOOL;
		oldTime : DINT;
		mappView : brdkViImg_mappView;
		imgArr : brdkVIImg_imageArray_typ;
		svgOverlay : STRING[5000];
		timeoutTrigger : TON;
		matchRes : ARRAY[0..19]OF pnp_vision_result_typ;
		rotPoint : brdkViBase_2d_typ;
		shapesPx : recipe_shapes_typ;
		getPicks : BOOL;
		mpRecipeRegPar : MpRecipeRegParSync;
	END_STRUCT;
	pnp_vision_results_shapeP_typ : 	STRUCT
		reference : ARRAY[0..MAX_SHAPE_POINTS]OF brdkViBase_2d_typ;
		clearenceStart : ARRAY[0..MAX_SHAPE_POINTS]OF brdkViBase_2d_typ;
		clearenceEnd : ARRAY[0..MAX_SHAPE_POINTS]OF brdkViBase_2d_typ;
	END_STRUCT;
	pnp_vision_result_typ : 	STRUCT
		pickPos : brdkViBase_3d_typ;
		imgPos : brdkViBase_2d_typ;
		ok : BOOL;
		angle : LREAL;
		shapePoints : pnp_vision_results_shapeP_typ;
	END_STRUCT;
	recipe_shapes_typ : 	STRUCT
		reference : brdkViGeom_shape_typ;
		clearenceStart : brdkViGeom_shape_typ;
		clearenceEnd : brdkViGeom_shape_typ;
	END_STRUCT;
	recipe_typ : 	STRUCT
		LEDsegment : USINT;
		focus : UINT; (*250*)
		expTime : DINT; (*50*)
		LED : USINT; (*1*)
		offset : brdkViBase_3d_typ;
		shapes : USINT;
		P : ARRAY[0..2,0..3]OF LREAL;
		imgQuality : USINT := 30;
		imgFormat : BRDKVIIMG_IMG_TYPE := BRDKVIIMG_IMG_TYPE_JPEG;
	END_STRUCT;
	va_res_typ : 	STRUCT
		numRes : USINT;
		res : ARRAY[0..19]OF blob_res_typ;
	END_STRUCT;
END_TYPE
```

#### Variables.var - Local variables
```iecst
VAR
	j : USINT;
	hw : cam_typ;
	state : USINT;
	hmi : hmi_typ;
	i : USINT;
	this : local_typ;
END_VAR
```

#### LightAction.st
```iecst
ACTION LightAction:

	 hw.out.angle[0]	:= REAL_TO_UINT(LIMIT(0,hmi.in.par.angle,135));
	hw.out.angle[1]		:= REAL_TO_UINT(LIMIT(0,180-hmi.in.par.angle,135));

	CASE state OF
		0:
			hmi.out.overlay1 := '';
			hmi.out.overlay2 := '';
			hmi.out.overlay3 := '';
			hmi.out.overlay4 := '';
			hmi.out.svg1 := '';
			hmi.out.svg2 := '';
			hmi.out.svg3 := '';
			hmi.out.svg4 := '';
			hmi.out.text1 := 'Front light';
			hmi.out.text2 := 'Backlight';

			state := 5;
		5:
			IF NOT hw.out.trigger  AND ((hw.in.ready[0] AND hw.in.ready[1] AND hw.in.ready[2] AND hw.in.ready[3]) OR DiagCpuIsSimulated()) AND this.mappView.status = ERR_OK THEN
				IF hmi.in.cmd.trigger THEN
					hmi.in.cmd.trigger := FALSE;
					state := 10;
					this.oldTime := hw.in.imgTime;
				END_IF
			END_IF

		10:
			// trigger image with nettime
			hw.out.trigger := TRUE;

			hw.out.enable := FALSE;
			hw.out.useRegionFeat := FALSE;

			hw.out.delayNettime := hw.in.nettime+ 20000;
			this.timeoutTrigger.PT := T#2000ms;
			this.timeoutTrigger.IN := TRUE;

			// Camera light only
			CASE hmi.in.par.LED[0] OF
				// 0 = none, 1= red, 2= green, 3= blue, 4=Lime, 5=White(99), 6=IR(100),7=UV(210)
				5:
					hw.out.ledColor[0] 	:= 99;
				6:
					hw.out.ledColor[0] 	:= 100;
				7:
					hw.out.ledColor[0] 	:= 210;
				ELSE
				hw.out.ledColor[0] 	:= hmi.in.par.LED[0];
			END_CASE

			hw.out.ledSegment 	:= 15;
			hw.out.expTime[0] 	:= hmi.in.par.expTime[0];

			hw.out.irFilter 	:= hw.out.ledColor[0] = 100;

			hw.out.ledColor[3] 	:= 0;
			hw.out.expTime[3] 	:= 0;

			hw.out.ledColor[2] 	:= 0;
			hw.out.expTime[2] 	:= 0;

			hw.out.ledColor[1] 	:= 0;
			hw.out.expTime[1]	:= 0;

			state := 20;

		20:
			// check if a new image is done
			IF hw.in.imgTime <> this.oldTime OR DiagCpuIsSimulated() THEN
				this.oldTime := hw.in.imgTime;
				this.mappView.updateImage := TRUE;
				this.mappView.pSvgImage 	:= ADR(hmi.out.svg1);
				hmi.in.cmd.trigger := FALSE;
				hw.out.trigger := FALSE;
				this.timeoutTrigger.IN := FALSE;

				state := 30;
			ELSIF this.timeoutTrigger.Q THEN
				state := 5;
				this.timeoutTrigger.IN := hw.out.trigger := FALSE;
				hmi.in.cmd.trigger := FALSE;
				hw.out.trigger := FALSE;
			END_IF

		30:
			this.TON_delay(IN := this.mappView.status = ERR_OK);

			IF (hw.in.ready[0] AND hw.in.ready[1] AND hw.in.ready[2] AND hw.in.ready[3]) AND this.TON_delay.Q THEN
				state := 40;
				this.TON_delay(IN := FALSE);
			END_IF

		40:
			// trigger image with nettime
			hw.out.trigger := TRUE;

			hw.out.enable := FALSE;
			hw.out.useRegionFeat := FALSE;

			hw.out.delayNettime := hw.in.nettime+ 20000;
			this.timeoutTrigger.PT := T#2000ms;
			this.timeoutTrigger.IN := TRUE;

			// Backlight only
			hw.out.ledColor[0] 	:= 0;
			hw.out.ledSegment 	:= 0;
			hw.out.expTime[0] 	:= hmi.in.par.expTime[0];

			hw.out.irFilter 	:= hw.out.ledColor[0] = 100;

			hw.out.ledColor[3] 	:= 0;
			hw.out.expTime[3] 	:= 0;

			hw.out.ledColor[2] 	:= 0;
			hw.out.expTime[2] 	:= 0;

			// Camera light only
			CASE hmi.in.par.LED[1] OF
				// 0 = none, 1= red, 2= green, 3= blue, 4=Lime, 5=White(99), 6=IR(100),7=UV(210)
				5:
					hw.out.ledColor[1] 	:= 99;
				6:
					hw.out.ledColor[1] 	:= 100;
				7:
					hw.out.ledColor[1] 	:= 210;
				ELSE
						hw.out.ledColor[1] 	:= hmi.in.par.LED[1];
			END_CASE

			hw.out.expTime[1]	:= hmi.in.par.expTime[1];

			state := 50;

		50:
			// check if a new image is done
			IF hw.in.imgTime <> this.oldTime OR DiagCpuIsSimulated() THEN
				this.oldTime := hw.in.imgTime;
				this.mappView.updateImage := TRUE;
				this.mappView.pSvgImage 	:= ADR(hmi.out.svg2);
				this.timeoutTrigger.IN := FALSE;

				hmi.in.cmd.trigger := FALSE;
				hw.out.trigger := FALSE;

				state := 60;
			ELSIF this.timeoutTrigger.Q THEN
				state := 5;
				this.timeoutTrigger.IN := hw.out.trigger := FALSE;
				hmi.in.cmd.trigger := FALSE;
				hw.out.trigger := FALSE;
			END_IF
		60:
			IF (hw.in.ready[0] AND hw.in.ready[1] AND hw.in.ready[2] AND hw.in.ready[3]) AND this.mappView.status = ERR_OK THEN
				state := 70;
			END_IF

		70:
			// trigger image with nettime
			hw.out.trigger := TRUE;

			hw.out.enable := FALSE;
			hw.out.useRegionFeat := FALSE;

			hw.out.delayNettime := hw.in.nettime+ 20000;
			this.timeoutTrigger.PT := T#2000ms;
			this.timeoutTrigger.IN := TRUE;

			// Barlights only
			hw.out.ledColor[0] 	:= 0;
			hw.out.ledSegment 	:= 0;
			hw.out.expTime[0] 	:= hmi.in.par.expTime[0];

			hw.out.irFilter 	:= hw.out.ledColor[0] = 100;

			hw.out.ledColor[1] 	:= 0;
			hw.out.expTime[1]	:= 0;

			CASE hmi.in.par.LED[2] OF
				// 0 = none, 1= red, 2= green, 3= blue, 4=Lime, 5=White(99), 6=IR(100),7=UV(210)
				5:
					hw.out.ledColor[2] 	:= 99;
				6:
					hw.out.ledColor[2] 	:= 100;
				7:
					hw.out.ledColor[2] 	:= 210;
				ELSE
						hw.out.ledColor[2] 	:= hmi.in.par.LED[2];
			END_CASE

			hw.out.expTime[3] := hw.out.expTime[2] 	:= hmi.in.par.expTime[2];
			hw.out.ledColor[3] 	:=hw.out.ledColor[2];

			state := 80;
		80:
			// check if a new image is done
			IF hw.in.imgTime <> this.oldTime OR DiagCpuIsSimulated() THEN
				this.oldTime := hw.in.imgTime;
				this.mappView.updateImage := TRUE;
				this.mappView.pSvgImage 	:= ADR(hmi.out.svg3);
				this.timeoutTrigger.IN := FALSE;

				hmi.in.cmd.trigger := FALSE;
				hw.out.trigger := FALSE;

				state := 90;
			ELSIF this.timeoutTrigger.Q THEN
				state := 5;
				this.timeoutTrigger.IN := hw.out.trigger := FALSE;
				hmi.in.cmd.trigger := FALSE;
				hw.out.trigger := FALSE;
			END_IF
		90:
			IF (hw.in.ready[0] AND hw.in.ready[1] AND hw.in.ready[2] AND hw.in.ready[3]) AND this.mappView.status = ERR_OK THEN
				state := 100;
			END_IF

		100:
			// trigger image with nettime
			hw.out.trigger := TRUE;

			hw.out.enable := FALSE;
			hw.out.useRegionFeat := FALSE;

			hw.out.delayNettime := hw.in.nettime+ 20000;
			this.timeoutTrigger.PT := T#2000ms;
			this.timeoutTrigger.IN := TRUE;

			// Backlight + barlights
			hw.out.ledColor[0] 	:= 0;
			hw.out.ledSegment 	:= 0;
			hw.out.expTime[0] 	:= hmi.in.par.expTime[0];

			hw.out.irFilter 	:= hw.out.ledColor[0] = 100;

			CASE hmi.in.par.LED[1] OF
				// 0 = none, 1= red, 2= green, 3= blue, 4=Lime, 5=White(99), 6=IR(100),7=UV(210)
				5:
					hw.out.ledColor[1] 	:= 99;
				6:
					hw.out.ledColor[1] 	:= 100;
				7:
					hw.out.ledColor[1] 	:= 210;
				ELSE
						hw.out.ledColor[1] 	:= hmi.in.par.LED[1];
			END_CASE
			hw.out.expTime[1]	:= hmi.in.par.expTime[1];

			CASE hmi.in.par.LED[2] OF
				// 0 = none, 1= red, 2= green, 3= blue, 4=Lime, 5=White(99), 6=IR(100),7=UV(210)
				5:
					hw.out.ledColor[2] 	:= 99;
				6:
					hw.out.ledColor[2] 	:= 100;
				7:
					hw.out.ledColor[2] 	:= 210;
				ELSE
						hw.out.ledColor[2] 	:= hmi.in.par.LED[2];
			END_CASE

			hw.out.expTime[3] := hw.out.expTime[2] 	:= hmi.in.par.expTime[2];
			hw.out.ledColor[3] 	:=hw.out.ledColor[2];

			state := 110;
		110:
			// check if a new image is done
			IF hw.in.imgTime <> this.oldTime OR DiagCpuIsSimulated() THEN
				this.oldTime := hw.in.imgTime;
				this.mappView.updateImage := TRUE;
				this.mappView.pSvgImage 	:= ADR(hmi.out.svg4);
				this.timeoutTrigger.IN := FALSE;

				hmi.in.cmd.trigger := FALSE;
				hw.out.trigger := FALSE;

				state := 5;
			ELSIF this.timeoutTrigger.Q THEN
				state := 5;
				this.timeoutTrigger.IN := hw.out.trigger := FALSE;
				hmi.in.cmd.trigger := FALSE;
				hw.out.trigger := FALSE;
			END_IF
	END_CASE
	this.timeoutTrigger();
END_ACTION
```

#### CalAction.st
```iecst
ACTION CalAction:

	CASE state OF
		0:
			IF NOT hw.out.trigger  AND (hw.in.ready[0] OR DiagCpuIsSimulated()) THEN
(*				IF hmi.in.cmd.calibrate THEN
					// for calibration we only look for 4 round Blobs

					state := 10;*)
				IF hmi.in.cmd.trigger THEN
					state := 10;
				END_IF
			END_IF

		10:
			// trigger image with nettime
			hw.out.trigger := TRUE;

			hw.out.numMax := 4;
			hw.out.enable := TRUE;
			hw.out.useRegionFeat := TRUE;

			hw.out.delayNettime := hw.in.nettime+ 20000;
			this.timeoutTrigger.PT := T#2000ms;
			this.timeoutTrigger.IN := TRUE;

			hw.out.ledColor[0] 	:= 0;
			hw.out.ledSegment 	:= hmi.in.par.LEDsegment;
			hw.out.expTime[0] 		:= hmi.in.par.expTime[0];

			hw.out.irFilter 	:= hw.out.ledColor[0] = 100;

			hw.out.ledColor[3] 	:= 0;
			hw.out.expTime[3] 	:= hmi.in.par.expTime[3];
			// TODO
			// hw.out.angle[1]		:=

			hw.out.ledColor[2] 	:= 0;
			hw.out.expTime[2] 	:= hmi.in.par.expTime[2];
			// TODO
			// hw.out.angle[0]		:=

			hw.out.ledColor[1] 	:= hmi.in.par.LED[1];
			hw.out.expTime[1]	:= hmi.in.par.expTime[1];

			state := 20;

		20:
			// check if a new image is done
			IF hw.in.imgTime <> this.oldTime OR DiagCpuIsSimulated() THEN
				this.oldTime := hw.in.imgTime;
				this.mappView.updateImage := TRUE;
				this.mappView.pSvgImage 	:= ADR(hmi.out.svg1);
				hmi.in.cmd.trigger := FALSE;
				hw.out.trigger := FALSE;

				IF hw.in.VA_match.numRes = 4 THEN
					state := 30;
				ELSE
					state := 0;
				END_IF
			ELSIF this.timeoutTrigger.Q THEN
				state := 0;
				this.timeoutTrigger.IN := hw.out.trigger := FALSE;
				hmi.in.cmd.trigger := FALSE;
				hw.out.trigger := FALSE;
			END_IF

		30:

				(*
	Calibation Plate

	|-------------------|
	|					| 37,5
	|	O			O	|
	|					| 			 150mm
	|					| 75mm
	|					|
	|	O		 	O	|
	| 					| 37,5mm
	--------------------|
	37,5     75mm    37,5
	_____________________
			150 mm

	Placement of real coordinate systems compared to image and calibration plate holes

	0,0         imgWidth,0
	   /|\ Y
	O	|	O
		|
	----------> X
		|
	O	|	O
		|
	0,imgHeiht	imgWidht,imgHeight
	*)

			FOR i:=0 TO 3 BY 1 DO
				this.imgPos[i].x := DINT_TO_LREAL(hw.in.va.res[i].posX) /100.0; // px
				this.imgPos[i].y := DINT_TO_LREAL(hw.in.va.res[i].posY) /100.0; // px

				IF this.imgPos[i].x > this.imgWidth/2 THEN
					this.realPos[i].x := 37.5; //mm
				ELSE
					this.realPos[i].x := -37.5; // mm

				END_IF

				IF this.imgPos[i].y > this.imgHeight/2 THEN
					this.realPos[i].y := -37.5; // mm

				ELSE
					this.realPos[i].y := 37.5; //mm
				END_IF

			END_FOR

			brdkViCal_Calibration(this.realPos[0],this.imgPos[0],4,hmi.in.par.P);

			hmi.out.overlay1 := '';
			brdkViGeom_drawCalibration(hmi.in.par.P,75,this.realPos[0],4,ADR(hmi.out.overlay1),ADR('style="fill:blue;stroke:blue;stroke-width:5;fill-opacity:0.3;stroke-opacity:1"'),ADR('style="fill:red;stroke:red;stroke-width:5;fill-opacity:1;stroke-opacity:1"'));
			state := 0;
	END_CASE

	// Handle image click event
	IF hmi.in.cmd.click THEN
		hmi.in.cmd.click := FALSE;

		this.tmp2D.x := hmi.in.cmd.x;
		this.tmp2D.y := hmi.in.cmd.y;

		// get invers projection matix (only need to be done one time as the projection matrix only changes if a new calibration is done
		brdkViCal_InvP(hmi.in.par.P,this.invP);

		// from image to real coordinates
		brdkViCal_2dTo3d(this.tmp2D,this.invP,hmi.out.realPos);

		hmi.out.overlay1 := '';
		this.tmp2D.x := this.tmp2D.x -50;
		this.tmp2D.y := this.tmp2D.y -50;

		brdkViGeom_drawSvgImage(ADR(this.url),this.tmp2D,ADR(''),100,100,ADR(hmi.out.overlay1),ADR(''));
		this.tmp2D.x := this.tmp2D.x +100;
		this.tmp2D.y := this.tmp2D.y +100;

	END_IF

	this.timeoutTrigger();
END_ACTION
```

#### ColAction.st
```iecst
ACTION ColAction:

	CASE state OF
		0:
			IF NOT hw.out.trigger  AND (hw.in.ready[0] OR DiagCpuIsSimulated()) THEN
				IF hmi.in.cmd.trigger THEN
					state := 10;
				END_IF
			END_IF

		10:
			// trigger image with nettime
			hw.out.trigger := TRUE;

			hw.out.enable := FALSE;
			hw.out.useRegionFeat := FALSE;

			hw.out.delayNettime := hw.in.nettime+ 20000;
			this.timeoutTrigger.PT := T#2000ms;
			this.timeoutTrigger.IN := TRUE;

			// Camera light only
			hw.out.ledColor[0] 	:= 1;
			hw.out.ledSegment 	:= hmi.in.par.LEDsegment;
			hw.out.expTime[0] 	:= hmi.in.par.expTime[0];

			hw.out.irFilter 	:= hw.out.ledColor[0] = 100;

			hw.out.ledColor[3] 	:= 0;
			hw.out.expTime[3] 	:= 0;

			hw.out.ledColor[2] 	:= 0;
			hw.out.expTime[2] 	:= 0;

			hw.out.ledColor[1] 	:= 0;
			hw.out.expTime[1]	:= 0;

			state := 20;

		20:
			// check if a new image is done
			IF hw.in.imgTime <> this.oldTime OR DiagCpuIsSimulated() THEN
				this.oldTime := hw.in.imgTime;
				this.mappView.updateImage := TRUE;

				hmi.in.cmd.trigger := FALSE;
				hw.out.trigger := FALSE;

				state := 30;
			ELSIF this.timeoutTrigger.Q THEN
				state := 0;
				this.timeoutTrigger.IN := hw.out.trigger := FALSE;
				hmi.in.cmd.trigger := FALSE;
				hw.out.trigger := FALSE;
			END_IF

		30:
			IF (hw.in.ready[0] AND hw.in.ready[1] AND hw.in.ready[2] AND hw.in.ready[3]) THEN
				state := 40;
			END_IF

		40:
			// trigger image with nettime
			hw.out.trigger := TRUE;

			hw.out.enable := FALSE;
			hw.out.useRegionFeat := FALSE;

			hw.out.delayNettime := hw.in.nettime+ 20000;
			this.timeoutTrigger.PT := T#2000ms;
			this.timeoutTrigger.IN := TRUE;

			// Camera light only
			hw.out.ledColor[0] 	:= 2;
			hw.out.ledSegment 	:= hmi.in.par.LEDsegment;
			hw.out.expTime[0] 	:= hmi.in.par.expTime[0];

			hw.out.irFilter 	:= hw.out.ledColor[0] = 100;

			hw.out.ledColor[3] 	:= 0;
			hw.out.expTime[3] 	:= 0;

			hw.out.ledColor[2] 	:= 0;
			hw.out.expTime[2] 	:= 0;

			hw.out.ledColor[1] 	:= 0;
			hw.out.expTime[1]	:= 0;

			state := 50;

		50:
			// check if a new image is done
			IF hw.in.imgTime <> this.oldTime OR DiagCpuIsSimulated() THEN
				this.oldTime := hw.in.imgTime;
				this.mappView.updateImage := TRUE;

				hmi.in.cmd.trigger := FALSE;
				hw.out.trigger := FALSE;

				state := 60;
			ELSIF this.timeoutTrigger.Q THEN
				state := 0;
				this.timeoutTrigger.IN := hw.out.trigger := FALSE;
				hmi.in.cmd.trigger := FALSE;
				hw.out.trigger := FALSE;
			END_IF
		60:
			IF (hw.in.ready[0] AND hw.in.ready[1] AND hw.in.ready[2] AND hw.in.ready[3]) THEN
				state := 70;
			END_IF

		70:
			// trigger image with nettime
			hw.out.trigger := TRUE;

			hw.out.enable := FALSE;
			hw.out.useRegionFeat := FALSE;

			hw.out.delayNettime := hw.in.nettime+ 20000;
			this.timeoutTrigger.PT := T#2000ms;
			this.timeoutTrigger.IN := TRUE;

			// Camera light only
			hw.out.ledColor[0] 	:= 3;
			hw.out.ledSegment 	:= hmi.in.par.LEDsegment;
			hw.out.expTime[0] 	:= hmi.in.par.expTime[0];

			hw.out.irFilter 	:= hw.out.ledColor[0] = 100;

			hw.out.ledColor[3] 	:= 0;
			hw.out.expTime[3] 	:= 0;

			hw.out.ledColor[2] 	:= 0;
			hw.out.expTime[2] 	:= 0;

			hw.out.ledColor[1] 	:= 0;
			hw.out.expTime[1]	:= 0;

			state := 80;
		80:
			// check if a new image is done
			IF hw.in.imgTime <> this.oldTime OR DiagCpuIsSimulated() THEN
				this.oldTime := hw.in.imgTime;
				this.mappView.updateImage := TRUE;

				hmi.in.cmd.trigger := FALSE;
				hw.out.trigger := FALSE;

				state := 90;
			ELSIF this.timeoutTrigger.Q THEN
				state := 0;
				this.timeoutTrigger.IN := hw.out.trigger := FALSE;
				hmi.in.cmd.trigger := FALSE;
				hw.out.trigger := FALSE;
			END_IF
		90:
			IF (hw.in.ready[0] AND hw.in.ready[1] AND hw.in.ready[2] AND hw.in.ready[3]) THEN
				state := 100;
			END_IF

		100:
			// trigger image with nettime
			hw.out.trigger := TRUE;

			hw.out.enable := FALSE;
			hw.out.useRegionFeat := FALSE;

			hw.out.delayNettime := hw.in.nettime+ 20000;
			this.timeoutTrigger.PT := T#2000ms;
			this.timeoutTrigger.IN := TRUE;

			// Camera light only
			hw.out.ledColor[0] 	:= 4;
			hw.out.ledSegment 	:= hmi.in.par.LEDsegment;
			hw.out.expTime[0] 	:= hmi.in.par.expTime[0];

			hw.out.irFilter 	:= hw.out.ledColor[0] = 100;

			hw.out.ledColor[3] 	:= 0;
			hw.out.expTime[3] 	:= 0;

			hw.out.ledColor[2] 	:= 0;
			hw.out.expTime[2] 	:= 0;

			hw.out.ledColor[1] 	:= 0;
			hw.out.expTime[1]	:= 0;

			state := 110;
		110:
			// check if a new image is done
			IF hw.in.imgTime <> this.oldTime OR DiagCpuIsSimulated() THEN
				this.oldTime := hw.in.imgTime;
				this.mappView.updateImage := TRUE;

				hmi.in.cmd.trigger := FALSE;
				hw.out.trigger := FALSE;

				state := 0;
			ELSIF this.timeoutTrigger.Q THEN
				state := 0;
				this.timeoutTrigger.IN := hw.out.trigger := FALSE;
				hmi.in.cmd.trigger := FALSE;
				hw.out.trigger := FALSE;
			END_IF
	END_CASE
	this.timeoutTrigger();

END_ACTION
```

#### MeasureAction.st
```iecst
ACTION MeasureAction:

END_ACTION
```

#### MatchAction.st
```iecst
ACTION MatchAction:

END_ACTION
```

#### OCRAction.st
```iecst
ACTION OCRAction:

END_ACTION
```

### Program Logical/Demo (IEC)

#### Main.st - Init, cyclic, exit code
```iecst
PROGRAM _INIT
	(* Insert code here *)
	// Init camera settings
	hmi.in.par.expTime := 700;
	hmi.in.par.focus := 411;
	hmi.in.par.LED := 1;
	hmi.in.par.LEDsegment := 15;

	this.mpRecipeRegPar.MpLink := ADR(gRecipeCsv);
	this.mpRecipeRegPar.PVName := ADR('::Demo:hmi.in.par');

END_PROGRAM

PROGRAM _CYCLIC

	CASE hmi.in.cmd.mode OF
		0: // Simple mode
			mainSimpleAction;
		1: // calibration Example
			mainCalibrationAction;

		2:
			mainColorAction;
	END_CASE

	this.viBaseSave(MpLink := ADR(gBlobCamera));
END_PROGRAM

PROGRAM _EXIT
	(* Insert code here *)
	this.mappView(enable := FALSE);
	this.getImage(enable := FALSE);
	this.mpRecipeRegPar(Enable := FALSE);

	IF this.wsServer.enable THEN
		FOR i := 0 TO UDINT_TO_USINT(BRDKVIIMG_WS_MAX_NUM_CLIENTS) BY 1 DO
			IF this.wsChannels[i].enable THEN
				this.wsChannels[i](enable 			:=  FALSE);
			END_IF
		END_FOR
		this.wsServer(enable := FALSE);

	END_IF

END_PROGRAM
```

#### Types.typ - Local data types
```iecst
TYPE
	match_res_typ : 	STRUCT
		score : USINT;
		angle : INT;
		posY : DINT;
		posX : DINT;
	END_STRUCT;
	blob_res_typ : 	STRUCT
		width : UDINT;
		maxX : DINT;
		minX : DINT;
		length : UDINT;
		posY : DINT;
		posX : DINT;
	END_STRUCT;
END_TYPE

(*Insert your comment here.*)

TYPE
	hmi_in_cmd_typ : 	STRUCT
		trigger : BOOL;
		calibrate : BOOL;
		elemId : STRING[80];
		y : REAL;
		x : REAL;
		click : BOOL;
		mode : USINT;
		useOPCua : BOOL := TRUE;
	END_STRUCT;
	hmi_in_typ : 	STRUCT
		cmd : hmi_in_cmd_typ;
		par : recipe_typ;
	END_STRUCT;
	hmi_out_color_typ : 	STRUCT
		red : STRING[6000000];
		green : STRING[6000000];
		blue : STRING[6000000];
	END_STRUCT;
	hmi_out_typ : 	STRUCT
		overlay : STRING[20000];
		svg : STRING[6000000];
		realPos : brdkViBase_3d_typ;
		pxColor : USINT;
		color : hmi_out_color_typ;
	END_STRUCT;
	hmi_typ : 	STRUCT
		in : hmi_in_typ;
		out : hmi_out_typ;
	END_STRUCT;
	hw_io_input_typ : 	STRUCT
		nettime : DINT;
	END_STRUCT;
	hw_io_typ : 	STRUCT
		input : hw_io_input_typ;
	END_STRUCT;
	hw_typ : 	STRUCT
		io : hw_io_typ;
		cam : brdkViBase_cam_hw_typ;
		backLight : ARRAY[0..0]OF brdkViBase_light_hw_typ;
		blob : brdkViBase_hw_blob_50_typ;
	END_STRUCT;
	local_tcpServer_typ : 	STRUCT
		clientIp : STRING[20];
		tcpSend : TcpSend;
	END_STRUCT;
	local_typ : 	STRUCT
		realPos : ARRAY[0..3]OF brdkViBase_3d_typ;
		imgPos : ARRAY[0..3]OF brdkViBase_2d_typ;
		invP : ARRAY[0..2,0..2]OF LREAL;
		imgCenter : brdkViBase_2d_typ;
		tmp2D1 : brdkViBase_2d_typ;
		tmp2D : brdkViBase_2d_typ;
		tmp3D : brdkViBase_3d_typ;
		tmpLREAL : LREAL;
		imgHeight : LREAL := 1024;
		imgWidth : LREAL := 1250;
		calcCalibrate : BOOL;
		oldTime : DINT;
		getImage : brdkViImg_getImage;
		mappView : brdkViImg_mappView;
		imgArr : brdkViImg_imageArray_typ;
		svgOverlay : STRING[5000];
		timeoutTrigger : TON;
		matchRes : ARRAY[0..19]OF pnp_vision_result_typ;
		rotPoint : brdkViBase_2d_typ;
		shapesPx : recipe_shapes_typ;
		getPicks : BOOL;
		mpRecipeRegPar : MpRecipeRegParSync;
		simFileDevice : STRING[10] := 'SIM';
		simFilename : STRING[100] := 'test';
		text : STRING[200] := 'this is a great test$NWith both new lines$N       and many white spaces';
		url : STRING[200] := 'Media/crossAir.png ';
		imgTrig : brdkViBase_imgTrigger;
		isCalibration : BOOL;
		cycleCnt : UDINT;
		sendBufLen : UDINT;
		tcpServer : local_tcpServer_typ;
		sendBuf : ARRAY[0..5000000]OF USINT;
		recvBuf : ARRAY[0..9999]OF USINT;
		wsRecData : ARRAY[0..BRDKVIIMG_WS_MAX_NUM_CLIENTS,0..199]OF USINT;
		wsChannels : ARRAY[0..BRDKVIIMG_WS_MAX_NUM_CLIENTS]OF brdkWS_Channel;
		wsServer : brdkWS_Server;
		wsSvg : STRING[6000000];
		viBaseSave : ViBaseSaveApplication;
	END_STRUCT;
	pnp_vision_results_shapeP_typ : 	STRUCT
		reference : ARRAY[0..MAX_SHAPE_POINTS]OF brdkViBase_2d_typ;
		clearenceStart : ARRAY[0..MAX_SHAPE_POINTS]OF brdkViBase_2d_typ;
		clearenceEnd : ARRAY[0..MAX_SHAPE_POINTS]OF brdkViBase_2d_typ;
	END_STRUCT;
	pnp_vision_result_typ : 	STRUCT
		pickPos : brdkViBase_3d_typ;
		imgPos : brdkViBase_2d_typ;
		ok : BOOL;
		angle : LREAL;
		shapePoints : pnp_vision_results_shapeP_typ;
	END_STRUCT;
	recipe_shapes_typ : 	STRUCT
		reference : brdkViGeom_shape_typ;
		clearenceStart : brdkViGeom_shape_typ;
		clearenceEnd : brdkViGeom_shape_typ;
	END_STRUCT;
	recipe_typ : 	STRUCT
		LEDsegment : USINT;
		focus : UINT; (*250*)
		expTime : DINT; (*50*)
		LED : USINT; (*1*)
		offset : brdkViBase_3d_typ;
		shapes : USINT;
		P : ARRAY[0..2,0..3]OF LREAL;
		imgQuality : USINT := 30;
		imgFormat : BRDKVIIMG_IMG_TYPE := BRDKVIIMG_IMG_TYPE_JPEG;
		wsPort : UINT := 18000;
	END_STRUCT;
	va_res_typ : 	STRUCT
		numRes : USINT;
		res : ARRAY[0..19]OF blob_res_typ;
	END_STRUCT;
	brdkViBase_hw_blob_50_in_typ : 	STRUCT  (*BLOB hardware input structure for 10 BLOB result*)
		common : brdkViBase_hw_vf_in_common_typ;
		results : ARRAY[0..49]OF brdkViBase_hw_blob_in_typ;
	END_STRUCT;
	brdkViBase_hw_blob_50_typ : 	STRUCT  (*BLOB hardware structure for 10 BLOB result*)
		in : brdkViBase_hw_blob_50_in_typ;
		out : brdkViBase_hw_blob_out_typ;
	END_STRUCT;
END_TYPE
```

#### Variables.var - Local variables
```iecst
VAR
	correcColor : ARRAY[0..2] OF REAL := [3(1)];
	j : USINT;
	clientIds : REFERENCE TO ARRAY[0..9] OF UDINT;
	hw : hw_typ;
	state : USINT;
	hmi : hmi_typ;
	i : USINT;
	this : local_typ;
END_VAR
```

#### MainSimpleAction.st - Init, cyclic, exit code
```iecst
ACTION mainSimpleAction:
	// always update pointers in case of copy download without execution of init/exit
	this.imgTrig.pCameraHw := ADR(hw.cam);
	this.imgTrig.pLightHw := ADR(hw.backLight);
	this.imgTrig.simulate.enable := DiagCpuIsSimulated();
	this.imgTrig.simulate.imgProcessingDelay := T#50ms;
	this.imgTrig.simulate.alwaysSimulateNonePresentLights := TRUE;
	this.imgTrig.simulate.alwaysSimulateNonePresentCamera := TRUE;

	// trigger image
	hw.cam.out.par.flashColor 	:= hmi.in.par.LED;
	hw.cam.out.par.flashSegment	:= hmi.in.par.LEDsegment;
	hw.cam.out.par.exposureTime	:= hmi.in.par.expTime;
	hw.cam.out.par.focus 		:= hmi.in.par.focus;
	hw.cam.out.par.IRFilter 	:= hw.cam.out.par.flashColor = BRDKVIBASE_CAM_LED_IR;

	// handles triggering af images
	this.imgTrig.pCameraHw := ADR(hw.cam); // Pointer to camera hw structure
	this.imgTrig.pLightHw := ADR(hw.backLight); // pointer to light structure or light structure array if more than one
	this.imgTrig.numLights := 1; //Number of lights
	this.imgTrig.useCamColorForLight := TRUE; // set Lights to same color as Camera
	this.imgTrig.useCamExpTimeForLight := TRUE; // Set light exposure time to same as camera
	this.imgTrig();

	// Trigger image
	IF this.imgTrig.ready AND NOT this.imgTrig.busy AND hmi.in.cmd.trigger THEN
		hmi.in.cmd.trigger 			:= FALSE;
		this.imgTrig.trigger 		:= TRUE;
		this.imgTrig.delayNettime 	:= hw.io.input.nettime + 50000; // add 50ms
	END_IF

	// Check for new image result
	IF this.imgTrig.newImage THEN
		this.mappView.updateImage := TRUE; // Trigger an update of the image on HMI

		IF hw.blob.in.common.numResults > 0 THEN
			FOR i:= 0 TO hw.blob.in.common.numResults-1 BY 1 DO
				this.tmp2D.x := DINT_TO_REAL(hw.blob.in.results[i].positionX) / 100.0;
				this.tmp2D.y := DINT_TO_REAL(hw.blob.in.results[i].positionY) / 100.0;
				// draw circle on overlay
				brdkViGeom_drawSvgCircle(this.tmp2D,50.0,ADR(hmi.out.overlay),ADR('style="fill:blue;stroke:blue;stroke-width:5;fill-opacity:0.3;stroke-opacity:1"'));

			END_FOR
		END_IF
	END_IF

	// Handle image click event on HMI image
	IF hmi.in.cmd.click THEN
		hmi.in.cmd.click := FALSE;

		this.tmp2D.x := hmi.in.cmd.x; //Click X coordinate
		this.tmp2D.y := hmi.in.cmd.y; // Click Y coordinate
		hmi.out.overlay := '';

		// If image is decoded and the size is larger than 0 then we can get the px value
		IF this.mappView.getImageArray AND 	this.imgArr.size > 0 THEN
			hmi.out.pxColor := brdkViImg_getPixel(LREAL_TO_INT(this.tmp2D.x),LREAL_TO_INT(this.tmp2D.y),this.imgArr.width,this.imgArr.pData); // Get pixel color value
		ELSE
			hmi.out.pxColor := 0;
		END_IF

		this.tmp2D.x := this.tmp2D.x -50; // offset -50 as image is 100 width such that center is in click position
		this.tmp2D.y := this.tmp2D.y -50; // offset -50 as image is 100 width such that center is in click position
		// Draw image in overlay (cross air)
		brdkViGeom_drawSvgImage(ADR(this.url),this.tmp2D,ADR(''),100,100,ADR(hmi.out.overlay),ADR(''));
	END_IF

	// Function to retrieve image from camera to show on HMI
	this.mappView.enable 		:= TRUE; // Enable
	this.mappView.pMappLink 	:= ADR(gBlobCamera); // Pointer to Vision component Mapp link variable
	this.mappView.getImageArray := TRUE; // If true the retrived image is also decoded to an USINT array
	this.mappView.pImageArray 	:= ADR(this.imgArr); // Pointer to brdkViImg_ImageArray_typ
	this.mappView.timeout 		:= 3000; // time out when retriving the image from the camera
	this.mappView.wsPort 		:= hmi.in.par.wsPort; // Web socket port number (use the same on brdk vision Image widget) (0 = web socket is not used)
	this.mappView.imageFormat 	:= hmi.in.par.imgFormat; // Image format to download JPEG or BMP
	this.mappView.jpegQuality 	:= hmi.in.par.imgQuality; // Quality for th	e JPEG image
	this.mappView.pImageArray 	:= ADR(this.imgArr); // Pointer to image array data structure (Decoded image information and 2d byte array)
	this.mappView.pSvgImage     := ADR(this.wsSvg); // Optional for web socket usage, but can be used to contain the SVG image if OPC UA is used
	// Simulation Configuration (Get images from file device instead of camera)
	this.mappView.simulateConfig.activate := DiagCpuIsSimulated(); // true if PLC is simulated
	this.mappView.simulateConfig.appendNumber := TRUE; // If true number is appended to file name
	this.mappView.simulateConfig.minNumber := 1; // Min number to append
	this.mappView.simulateConfig.maxNumber := 3; // Max number to append
	this.mappView.simulateConfig.autoIncrementNumber := TRUE; // Automatically Increment number
	this.mappView.simulateConfig.pDevice := ADR(this.simFileDevice); // Pointer to file device name where simulation images are located
	this.mappView.simulateConfig.pFile := ADR(this.simFilename); // pointer to filename string (with out file extension, which come from seleted image type Jpeg or BMP) where number is appended to
	this.mappView();

	this.getImage(enable := FALSE); // not used as the one inside mappView is used
	this.wsServer(enable := FALSE); // not used as the one inside mappView is used

	// recipe
	this.mpRecipeRegPar.ConfirmSave := this.mpRecipeRegPar.SaveNotification;
	this.mpRecipeRegPar(Enable := TRUE);

END_ACTION
```

#### MainCalibrationAction.st
```iecst
ACTION	mainCalibrationAction:
	// always update pointers in case of copy download without execution of init/exit
	this.imgTrig.pCameraHw := ADR(hw.cam);
	this.imgTrig.pLightHw := ADR(hw.backLight);

	// trigger image
	hw.cam.out.par.flashColor 	:= hmi.in.par.LED;
	hw.cam.out.par.flashSegment	:= hmi.in.par.LEDsegment;
	hw.cam.out.par.exposureTime	:= hmi.in.par.expTime;
	hw.cam.out.par.focus 		:= hmi.in.par.focus;
	hw.cam.out.par.IRFilter 	:= hw.cam.out.par.flashColor = BRDKVIBASE_CAM_LED_IR;

	IF hmi.in.cmd.calibrate THEN
		// for calibration we only look for 4 round Blobs
		hw.blob.out.common.numSearchMax := 4;
		hw.blob.out.common.enable := TRUE;
		hw.blob.out.regionFeatures := TRUE;
	ELSIF hmi.in.cmd.trigger THEN
		hw.blob.out.common.enable := FALSE;
		hw.blob.out.regionFeatures := FALSE;
	END_IF

	// handles triggering af images
	this.imgTrig.pLightHw := ADR(hw.backLight); // pointer to light structure or light structure array if more than one
	this.imgTrig.numLights := 1; //Number of lights
	this.imgTrig.useCamColorForLight := TRUE; // set Lights to same color as Camera
	this.imgTrig.useCamExpTimeForLight := TRUE; // Set light exposure time to same as camera
	this.imgTrig();

	// IF calibration then also trigger an image
	IF EDGEPOS(hmi.in.cmd.calibrate) THEN
		hmi.in.cmd.trigger := TRUE;
	END_IF

	// Trigger image
	IF ((this.imgTrig.ready AND NOT this.imgTrig.busy) OR DiagCpuIsSimulated()) AND hmi.in.cmd.trigger THEN
		hmi.in.cmd.trigger 			:= FALSE;
		this.imgTrig.trigger 		:= TRUE;
		this.imgTrig.delayNettime 	:= hw.io.input.nettime + 50000; // add 50ms
	END_IF

	// Check for new image result
	IF this.imgTrig.newImage OR (this.imgTrig.trigger AND DiagCpuIsSimulated()) THEN
		this.mappView.updateImage := TRUE;

		// incase of simulation hardware results
		IF DiagCpuIsSimulated() THEN
			// Random error
			IF brdkViBase_random(0,7) > 4 THEN
				hw.blob.in.common.numResults := 3;
			ELSE
				hw.blob.in.common.numResults := 4;
			END_IF

			hw.blob.in.results[0].positionX := 31118;
			hw.blob.in.results[0].positionY := 15084;
			hw.blob.in.results[1].positionX := 74896;
			hw.blob.in.results[1].positionY := 15408;
			hw.blob.in.results[2].positionX := 31487;
			hw.blob.in.results[2].positionY := 58665;
			hw.blob.in.results[3].positionX := 74391;
			hw.blob.in.results[3].positionY := 58582;
		END_IF

		// check if its a calibration or its a pick result image
		IF hmi.in.cmd.calibrate THEN
			this.mappView.simulateConfig.maxNumber := 1; // select only first image

			IF hw.blob.in.common.numResults = 4 THEN
			(*
				Calibation Plate

				|-------------------|
				|					| 37,5
				|	O			O	|
				|					| 			 150mm
				|					| 75mm
				|					|
				|	O		 	O	|
				| 					| 37,5mm
				--------------------|
				37,5     75mm    37,5
				_____________________
						150 mm

				Placement of real coordinate systems compared to image and calibration plate holes

				0,0         imgWidth,0
				   /|\ Y
				O	|	O
					|
				----------> X
					|
				O	|	O
					|
				0,imgHeiht	imgWidht,imgHeight
			*)

			// Transfer VA results to 2 image points
				FOR i:=0 TO 3 BY 1 DO
					// if simulation then fill in four points

					// scale to px decimal value
					this.imgPos[i].x := DINT_TO_REAL(hw.blob.in.results[i].positionX) / 100.0;
					this.imgPos[i].y := DINT_TO_REAL(hw.blob.in.results[i].positionY) / 100.0;

					// Hardcoded check for point location in each quater of the image
					IF this.imgPos[i].x > this.imgWidth/2 THEN
						this.realPos[i].x := 37.5; //mm
					ELSE
						this.realPos[i].x := -37.5; // mm

					END_IF

					IF this.imgPos[i].y > this.imgHeight/2 THEN
						this.realPos[i].y := -37.5; // mm

					ELSE
						this.realPos[i].y := 37.5; //mm
					END_IF

				END_FOR

				// Calculate camera projection matrix (3d -> img coordinate) based on four 3D points the four corresponding img points
				brdkViCal_Calibration(this.realPos[0],this.imgPos[0],4,hmi.in.par.P);

				// get invers projection matix (only need to be done one time as the projection matrix only changes if a new calibration is done
				brdkViCal_InvP(hmi.in.par.P,this.invP);

				hmi.out.overlay := ''; // Clear overlay
				// Draw the calibration result based on the 3D data (the four points and x and y axis )
				brdkViGeom_drawCalibration(hmi.in.par.P,75,this.realPos[0],4,10,ADR(hmi.out.overlay),ADR('style="fill:blue;stroke:blue;stroke-width:5;fill-opacity:0.3;stroke-opacity:1"'),ADR('style="fill:red;stroke:red;stroke-width:5;fill-opacity:1;stroke-opacity:1"'));

			ELSE // if numresults <> 4
				hmi.out.overlay := ''; // Clear overlay

				// Draw warning text on image
				this.tmp2D.x := 50;
				this.tmp2D.y := 50;
				brdkViGeom_drawSvgText(ADR('Warning: The four point BLOBs was not found!!$N check MappVision for model details.'),this.tmp2D,1,ADR(hmi.out.overlay),ADR('style="font: italic 40px serif; fill: red;"'));

				// Draw the found results
				IF hw.blob.in.common.numResults > 0 THEN
					FOR i:=0 TO hw.blob.in.common.numResults-1 BY 1 DO
						// Draw circle
						this.tmp2D.x := DINT_TO_REAL(hw.blob.in.results[i].positionX) / 100.0;
						this.tmp2D.y := DINT_TO_REAL(hw.blob.in.results[i].positionY) / 100.0;
						brdkViGeom_drawSvgCircle(this.tmp2D,50.0,ADR(hmi.out.overlay),ADR('style="fill:blue;stroke:red;stroke-width:5;fill-opacity:0.3;stroke-opacity:1"'));
					END_FOR
				END_IF
			END_IF // END if numResults = 4
		ELSE // If not calibrate, Process found results
			this.mappView.simulateConfig.maxNumber := 3; // reset to 3 as calibrate might have set it to 1

			// reset current results
			brsmemset(ADR(this.matchRes),0,SIZEOF(this.matchRes));
			hmi.out.overlay := '';

			// Process each result from the VF
			FOR i:= 0 TO hw.blob.in.common.numResults BY 1 DO

				// convert to decimal numbers (and offset andge)
				this.matchRes[i].imgPos.x := DINT_TO_REAL(hw.blob.in.results[i].positionX) / 100.0;
				this.matchRes[i].imgPos.y := DINT_TO_REAL(hw.blob.in.results[i].positionY) / 100.0;
				this.matchRes[i].angle := DINT_TO_REAL(hw.blob.in.results[i].orientation) / 100.0 + hmi.in.par.offset.z;

				// find rotation point (will be used to add offset to x and y axis relative to object orientation)
				this.rotPoint.x := COS(this.matchRes[i].angle*0.0174532925199444);
				this.rotPoint.y := SIN(this.matchRes[i].angle*-0.0174532925199444);
				// add offset (x,y) to object poisition relative to object orientation
				this.matchRes[i].imgPos.x := this.matchRes[i].imgPos.x  + this.rotPoint.x*hmi.in.par.offset.x + this.rotPoint.y*hmi.in.par.offset.y;
				this.matchRes[i].imgPos.y := this.matchRes[i].imgPos.y  + this.rotPoint.y*hmi.in.par.offset.x - this.rotPoint.x*hmi.in.par.offset.y;

				// Get 3d position
				brdkViCal_2dTo3d(this.matchRes[i].imgPos,this.invP,this.matchRes[i].pickPos); // Project px to mm
				this.matchRes[i].pickPos.z := LREAL_TO_REAL(brdkViCal_2dto3dOrientation(this.matchRes[i].angle,this.invP,this.imgCenter.x,this.imgCenter.y));

				// offset shape point to result location
				IF this.shapesPx.clearenceEnd.numPoints > 0 THEN
					FOR j:=0 TO this.shapesPx.clearenceEnd.numPoints - 1 BY 1 DO
						brdkViGeom_offsetVector(-this.matchRes[i].angle, this.matchRes[i].imgPos,this.matchRes[i].shapePoints.clearenceEnd[j]);
					END_FOR
					brdkViGeom_drawSvgPoly(this.matchRes[i].shapePoints.clearenceEnd[0],this.shapesPx.clearenceEnd.numPoints, ADR(hmi.out.overlay),ADR('style="fill:yellow;stroke:yellow;stroke-width:5;fill-opacity:0.3;stroke-opacity:1"'));
				END_IF

				IF this.shapesPx.clearenceStart.numPoints > 0 THEN
					FOR j:=0 TO this.shapesPx.clearenceStart.numPoints - 1 BY 1 DO
						brdkViGeom_offsetVector(-this.matchRes[i].angle, this.matchRes[i].imgPos,this.matchRes[i].shapePoints.clearenceStart[j]);
					END_FOR
					brdkViGeom_drawSvgPoly(this.matchRes[i].shapePoints.clearenceStart[0],this.shapesPx.clearenceStart.numPoints, ADR(hmi.out.overlay),ADR('style="fill:yellow;stroke:yellow;stroke-width:5;fill-opacity:0.3;stroke-opacity:1"'));
				END_IF

				IF this.shapesPx.reference.numPoints > 0 THEN
					FOR j:=0 TO this.shapesPx.reference.numPoints - 1 BY 1 DO
						brdkViGeom_offsetVector(-this.matchRes[i].angle, this.matchRes[i].imgPos,this.matchRes[i].shapePoints.reference[j]);
					END_FOR
					brdkViGeom_drawSvgPoly(this.matchRes[i].shapePoints.reference[0],this.shapesPx.reference.numPoints, ADR(hmi.out.overlay),ADR('style="fill:green;stroke:green;stroke-width:5;fill-opacity:0.3;stroke-opacity:1"'));
				END_IF
			END_FOR
		END_IF
	END_IF // end New image results

	// Handle image click event
	IF hmi.in.cmd.click THEN
		hmi.in.cmd.click := FALSE;

		this.tmp2D.x := hmi.in.cmd.x;
		this.tmp2D.y := hmi.in.cmd.y;

		// If image is decoded and the size is larger than 0 then we can get the px value
		IF this.mappView.getImageArray AND 	this.imgArr.size > 0 THEN
			hmi.out.pxColor := brdkViImg_getPixel(LREAL_TO_INT(this.tmp2D.x),LREAL_TO_INT(this.tmp2D.y),this.imgArr.width,this.imgArr.pData); // Get pixel color value
		ELSE
			hmi.out.pxColor := 0;
		END_IF

		//convert click image coordiantes to real coordinates
		brdkViCal_2dTo3d(this.tmp2D,this.invP,hmi.out.realPos);

		hmi.out.overlay := '';
		this.tmp2D.x := this.tmp2D.x -50;
		this.tmp2D.y := this.tmp2D.y -50;

		brdkViGeom_drawSvgImage(ADR(this.url),this.tmp2D,ADR(''),100,100,ADR(hmi.out.overlay),ADR(''));
	END_IF

	this.mappView.wsPort 		:= 18001;
	this.mappView.imageFormat 	:= hmi.in.par.imgFormat;
	this.mappView.jpegQuality 	:= hmi.in.par.imgQuality;
	this.mappView.pSvgImage 	:= 0;//ADR(hmi.out.svg);
	this.mappView.pImageArray 	:= ADR(this.imgArr);
	// Simulation Configuration (Get images from file device instead of camera)
	this.mappView.simulateConfig.activate := DiagCpuIsSimulated(); // true if PLC is simulated
	this.mappView.simulateConfig.appendNumber := TRUE; // If true number is appended to file name
	this.mappView.simulateConfig.minNumber := 1; // Min number to append
	this.mappView.simulateConfig.maxNumber := 3; // Max number to append
	this.mappView.simulateConfig.autoIncrementNumber := TRUE; // Automatically Increment number
	this.mappView.simulateConfig.pDevice := ADR(this.simFileDevice); // Pointer to file device name where simulation images are located
	this.mappView.simulateConfig.pFile := ADR(this.simFilename); // pointer to filename string (with out file extension, which come from seleted image type Jpeg or BMP) where number is appended to
	this.mappView();

	this.getImage(enable := FALSE); // not used as the one inside mappView is used
	this.wsServer(enable := FALSE); // not used as the one inside mappView is used

	// recipe
	this.mpRecipeRegPar.ConfirmSave := this.mpRecipeRegPar.SaveNotification;
	this.mpRecipeRegPar(Enable := TRUE);

END_ACTION
```

#### MainColorAction.st - Init, cyclic, exit code
```iecst
ACTION mainColorAction:
	// always update pointers in case of copy download without execution of init/exit
	this.imgTrig.pCameraHw := ADR(hw.cam);
	this.imgTrig.pLightHw := 0;
	this.imgTrig.numLights := 0;
	this.getImage.timeout := t#1s;
	// trigger image
	hw.cam.out.par.flashSegment	:= hmi.in.par.LEDsegment;
	hw.cam.out.par.focus 		:= hmi.in.par.focus;
	hw.cam.out.par.IRFilter 	:= hw.cam.out.par.flashColor = BRDKVIBASE_CAM_LED_IR;

	// handles triggering af images
	this.imgTrig.pLightHw := ADR(hw.backLight); // pointer to light structure or light structure array if more than one
	this.imgTrig.numLights := 1; //Number of lights
	this.imgTrig.useCamColorForLight := TRUE; // set Lights to same color as Camera
	this.imgTrig.useCamExpTimeForLight := TRUE; // Set light exposure time to same as camera
	this.imgTrig();

	// Check for new image result
	IF this.imgTrig.newImage OR (this.imgTrig.trigger AND DiagCpuIsSimulated()) THEN
		this.getImage.getImage := TRUE; // Trigger an update of the image on HMI
	END_IF

	IF state > 0 AND state < 120  THEN
		this.cycleCnt := this.cycleCnt+1;
	END_IF

	CASE state OF
		0:

			IF ((this.imgTrig.ready AND NOT this.imgTrig.busy) OR DiagCpuIsSimulated()) AND hmi.in.cmd.trigger THEN // camera is ready for new trigger
				this.cycleCnt := 0;
				hmi.in.cmd.trigger 			:= FALSE;
				this.imgTrig.trigger 		:= TRUE;
				hw.cam.out.par.flashColor 	:= BRDKVIBASE_CAM_LED_RED;
				hw.cam.out.par.exposureTime	:= REAL_TO_UDINT(UDINT_TO_REAL(brdkViBase_LEDIntensity(2, hmi.in.par.focus, hmi.in.par.expTime,BRDKVIBASE_CAM_LED_RED,BRDKVIBASE_CAM_LED_RED))*correcColor[0]); //;
				this.imgTrig.delayNettime 	:= hw.io.input.nettime + 8000; // add 50ms
				state := 10;

			END_IF

		10:
			IF this.getImage.getImage THEN // image have been caputured and download has begun

				state := 20;
			END_IF

		20:
			IF this.getImage.status = ERR_OK THEN // Image download from camera has finished
				this.sendBufLen := 0; // Clear frame for new
				brdkWS_MakeFrame(ADR('RED'),3,ADR(this.sendBuf),ADR(this.sendBufLen),TRUE);
				brdkWS_MakeFrame(this.getImage.pDest,this.getImage.destLen ,ADR(this.sendBuf),ADR(this.sendBufLen),FALSE);
				state := 100;
			ELSIF this.getImage.status = ERR_BRDKVIIMG_NO_IMAGE THEN
				this.imgTrig.trigger 		:= TRUE;
				hw.cam.out.par.flashColor 	:= BRDKVIBASE_CAM_LED_RED;
				hw.cam.out.par.exposureTime	:= REAL_TO_UDINT(UDINT_TO_REAL(brdkViBase_LEDIntensity(2, hmi.in.par.focus, hmi.in.par.expTime,BRDKVIBASE_CAM_LED_RED,BRDKVIBASE_CAM_LED_RED))*correcColor[0]); //;
				this.imgTrig.delayNettime 	:= hw.io.input.nettime + 8000; // add 50ms

				state := 10;
			END_IF
		100:

			IF ((this.imgTrig.ready AND NOT this.imgTrig.busy) OR DiagCpuIsSimulated()) THEN
				hmi.in.cmd.trigger 			:= FALSE;
				this.imgTrig.trigger 		:= TRUE;
				hw.cam.out.par.exposureTime	:= REAL_TO_UDINT(UDINT_TO_REAL(brdkViBase_LEDIntensity(2, hmi.in.par.focus, hmi.in.par.expTime,BRDKVIBASE_CAM_LED_RED,BRDKVIBASE_CAM_LED_GREEN))*correcColor[1]);
				hw.cam.out.par.flashColor 	:= BRDKVIBASE_CAM_LED_GREEN;
				this.imgTrig.delayNettime 	:= hw.io.input.nettime + 8000; // add 50ms
				state := 110;
			END_IF

		110:
			IF this.getImage.getImage THEN
				state := 115;
			END_IF
		115:

			IF this.getImage.status = ERR_OK THEN

				brdkWS_MakeFrame(ADR('Green'),5,ADR(this.sendBuf),ADR(this.sendBufLen),TRUE);
				brdkWS_MakeFrame(this.getImage.pDest,this.getImage.destLen ,ADR(this.sendBuf),ADR(this.sendBufLen),FALSE);

				state := 120;
//				IF this.getImage.getImage THEN
//					state := 220;
//				ELSE
//					state := 200;
//				END_IF
			ELSIF this.getImage.status = ERR_BRDKVIIMG_NO_IMAGE THEN
				this.imgTrig.trigger 		:= TRUE;
				hw.cam.out.par.exposureTime	:= REAL_TO_UDINT(UDINT_TO_REAL(brdkViBase_LEDIntensity(2, hmi.in.par.focus, hmi.in.par.expTime,BRDKVIBASE_CAM_LED_RED,BRDKVIBASE_CAM_LED_GREEN))*correcColor[1]);
				hw.cam.out.par.flashColor 	:= BRDKVIBASE_CAM_LED_GREEN;
				this.imgTrig.delayNettime 	:= hw.io.input.nettime + 8000; // add 50ms

				state := 100;
			END_IF
		120:
			IF ((this.imgTrig.ready AND NOT this.imgTrig.busy) OR DiagCpuIsSimulated()) THEN
				hmi.in.cmd.trigger 			:= FALSE;
				this.imgTrig.trigger 		:= TRUE;
				hw.cam.out.par.exposureTime	:= REAL_TO_UDINT(UDINT_TO_REAL(brdkViBase_LEDIntensity(2, hmi.in.par.focus, hmi.in.par.expTime,BRDKVIBASE_CAM_LED_RED,BRDKVIBASE_CAM_LED_BLUE))*correcColor[2]);
				hw.cam.out.par.flashColor 	:= BRDKVIBASE_CAM_LED_BLUE;
				this.imgTrig.delayNettime 	:= hw.io.input.nettime + 8000; // add 50ms
				state := 200;
			END_IF

		200:
			IF this.getImage.getImage THEN
				state := 220;
			END_IF

		220:
			IF this.getImage.status = ERR_OK AND NOT this.tcpServer.tcpSend.enable THEN
					state := 0;

					brdkWS_MakeFrame(ADR('BLUE'),4,ADR(this.sendBuf),ADR(this.sendBufLen),TRUE);
					brdkWS_MakeFrame(this.getImage.pDest,this.getImage.destLen ,ADR(this.sendBuf),ADR(this.sendBufLen),FALSE);
					brdkWS_MakeFrame(ADR('Done'),4,ADR(this.sendBuf),ADR(this.sendBufLen),TRUE);

					FOR i :=0 TO UDINT_TO_USINT(BRDKVIIMG_WS_MAX_NUM_CLIENTS) BY 1 DO
						IF this.wsChannels[i].enable THEN
							this.wsChannels[i].pSendData 	:= ADR(this.sendBuf);
							this.wsChannels[i].sendLen 		:= this.sendBufLen;
							this.wsChannels[i].doSend 		:= TRUE;
							END_IF
					END_FOR

			ELSIF this.getImage.status = ERR_BRDKVIIMG_NO_IMAGE THEN

				this.imgTrig.trigger 		:= TRUE;
				hw.cam.out.par.exposureTime	:= REAL_TO_UDINT(UDINT_TO_REAL(brdkViBase_LEDIntensity(2, hmi.in.par.focus, hmi.in.par.expTime,BRDKVIBASE_CAM_LED_RED,BRDKVIBASE_CAM_LED_BLUE))*correcColor[2]);
				hw.cam.out.par.flashColor 	:= BRDKVIBASE_CAM_LED_BLUE;
				this.imgTrig.delayNettime 	:= hw.io.input.nettime + 8000; // add 50ms
				state := 200;

			END_IF
	END_CASE
	//

	this.wsServer.enable := TRUE;
	this.wsServer.pIfAddr := 0;
	this.wsServer.port := 18070;
	this.wsServer();

	IF this.wsServer.enable THEN
		FOR i := 0 TO UDINT_TO_USINT(BRDKVIIMG_WS_MAX_NUM_CLIENTS) BY 1 DO
			IF this.wsServer.clients[i] <> 0 THEN
				this.wsChannels[i].enable 			:=  TRUE;
				this.wsChannels[i].ident 			:= this.wsServer.clients[i];
				this.wsChannels[i].bufferSize 		:= BRDKVIIMG_WS_BUFFER_SIZE;
				this.wsChannels[i].parentServer 	:= ADR(this.wsServer);
				this.wsChannels[i].pRecvData 		:= ADR(this.wsRecData[i,0]);
			ELSE
				this.wsChannels[i].enable 			:=  FALSE;
			END_IF
			this.wsChannels[i]();

		END_FOR
	END_IF

	// Function to retrieve image from camera to show on HMI
	this.getImage.enable := TRUE;
	this.getImage.pMappLink := ADR(gBlobCamera);
	this.getImage.imageFormat 	:= hmi.in.par.imgFormat;
	this.getImage.jpegQuality 	:= hmi.in.par.imgQuality;
	this.getImage.simulateConfig.activate := DiagCpuIsSimulated(); // true if PLC is simulated
	this.getImage.simulateConfig.appendNumber := TRUE; // If true number is appended to file name
	this.getImage.simulateConfig.minNumber := 1; // Min number to append
	this.getImage.simulateConfig.maxNumber := 3; // Max number to append
	this.getImage.simulateConfig.autoIncrementNumber := TRUE; // Automatically Increment number
	this.getImage.simulateConfig.pDevice := ADR(this.simFileDevice); // Pointer to file device name where simulation images are located
	this.getImage.simulateConfig.pFile := ADR(this.simFilename); // pointer to filename string (with out file extension, which come from seleted image type Jpeg or BMP) where number is appended to
	this.getImage();

	this.mappView(enable := FALSE); // Do not use as we get the images with getImage and send them as binary with wsServer and brdkWS_MakeFrame

	// recipe
	this.mpRecipeRegPar.ConfirmSave := this.mpRecipeRegPar.SaveNotification;
	this.mpRecipeRegPar(Enable := TRUE);

END_ACTION
```
